LIN {X 0,Y 490.317,Z 298.891,A -85,B 0,C 180,E1 -6360.634,E2 -6360.634} C_VEL
LIN {X 0,Y 489.99,Z 352.828,A -85,B 0,C 180,E1 -6361.447,E2 -6361.447} C_VEL
LIN {X 0,Y 489.88,Z 362.097,A -85,B 0,C 180,E1 -6361.688,E2 -6361.688} C_VEL
LIN {X 0,Y 489.724,Z 372.302,A -85,B 0,C 180,E1 -6362.083,E2 -6362.083} C_VEL
LIN {X 0,Y 489.479,Z 384.149,A -85,B 0,C 180,E1 -6362.737,E2 -6362.737} C_VEL
LIN {X 0,Y 489.252,Z 392.699,A -85,B 0,C 180,E1 -6363.367,E2 -6363.367} C_VEL
LIN {X 0,Y 488.984,Z 399.772,A -85,B 0,C 180,E1 -6364,E2 -6364} C_VEL
LIN {X 0,Y 488.756,Z 406.629,A -85,B 0,C 180,E1 -6364.743,E2 -6364.743} C_VEL
LIN {X 0,Y 488.57,Z 412.949,A -85,B 0,C 180,E1 -6365.571,E2 -6365.571} C_VEL
LIN {X 0,Y 488.385,Z 418.571,A -85,B 0,C 180,E1 -6366.464,E2 -6366.464} C_VEL
LIN {X 0,Y 488.232,Z 423.172,A -85,B 0,C 180,E1 -6367.353,E2 -6367.353} C_VEL
LIN {X 0,Y 488.108,Z 427.721,A -85,B 0,C 180,E1 -6368.46,E2 -6368.46} C_VEL
LIN {X 0,Y 488.055,Z 430.624,A -85,B 0,C 180,E1 -6369.377,E2 -6369.377} C_VEL
LIN {X 0,Y 487.919,Z 433.524,A -85,B 0,C 180,E1 -6370.653,E2 -6370.653} C_VEL
LIN {X 0,Y 487.896,Z 435.193,A -85,B 0,C 180,E1 -6371.921,E2 -6371.921} C_VEL
LIN {X 0,Y 487.875,Z 435.589,A -85,B 0,C 180,E1 -6373.256,E2 -6373.256} C_VEL
LIN {X 0,Y 487.923,Z 435.219,A -85,B 0,C 180,E1 -6374.117,E2 -6374.117} C_VEL
LIN {X 0,Y 487.927,Z 434.243,A -85,B 0,C 180,E1 -6374.973,E2 -6374.973} C_VEL
LIN {X 0,Y 487.992,Z 431.831,A -85,B 0,C 180,E1 -6376.253,E2 -6376.253} C_VEL
LIN {X 0,Y 488.088,Z 428.018,A -85,B 0,C 180,E1 -6377.527,E2 -6377.527} C_VEL
LIN {X 0,Y 488.18,Z 424.744,A -85,B 0,C 180,E1 -6378.373,E2 -6378.373} C_VEL
LIN {X 0,Y 488.358,Z 419.564,A -85,B 0,C 180,E1 -6379.427,E2 -6379.427} C_VEL
LIN {X 0,Y 488.473,Z 414.514,A -85,B 0,C 180,E1 -6380.267,E2 -6380.267} C_VEL
LIN {X 0,Y 488.635,Z 408.418,A -85,B 0,C 180,E1 -6381.106,E2 -6381.106} C_VEL
LIN {X 0,Y 488.95,Z 401.875,A -85,B 0,C 180,E1 -6381.85,E2 -6381.85} C_VEL
LIN {X 0,Y 489.127,Z 394.255,A -85,B 0,C 180,E1 -6382.57,E2 -6382.57} C_VEL
LIN {X 0,Y 489.382,Z 386.064,A -85,B 0,C 180,E1 -6383.198,E2 -6383.198} C_VEL
LIN {X 0,Y 489.583,Z 377.622,A -85,B 0,C 180,E1 -6383.716,E2 -6383.716} C_VEL
LIN {X 0,Y 489.769,Z 367.721,A -85,B 0,C 180,E1 -6384.184,E2 -6384.184} C_VEL
LIN {X 0,Y 489.927,Z 355.422,A -85,B 0,C 180,E1 -6384.573,E2 -6384.573} C_VEL
LIN {X 0,Y 490.062,Z 334.881,A -85,B 0,C 180,E1 -6384.909,E2 -6384.909} C_VEL
LIN {X 0,Y 490.212,Z 286.553,A -85,B 0,C 180,E1 -6385.619,E2 -6385.619} C_VEL
LIN {X 0,Y 488.623,Z 277.035,A -85,B 0,C 180,E1 -6385.824,E2 -6385.824} C_VEL
LIN {X 0,Y 488.729,Z 264.417,A -85,B 0,C 180,E1 -6388.764,E2 -6388.764} C_VEL
LIN {X 0,Y 488.756,Z 259.415,A -85,B 0,C 180,E1 -6389.949,E2 -6389.949} C_VEL
LIN {X 0,Y 488.939,Z 259.395,A -85,B 0,C 180,E1 -6390.824,E2 -6390.824} C_VEL
LIN {X 0,Y 488.921,Z 259.391,A -85,B 0,C 180,E1 -6392.472,E2 -6392.472} C_VEL
LIN {X 0,Y 488.816,Z 259.406,A -85,B 0,C 180,E1 -6395.776,E2 -6395.776} C_VEL
LIN {X 0,Y 488.778,Z 259.408,A -85,B 0,C 180,E1 -6398.267,E2 -6398.267} C_VEL
LIN {X 0,Y 488.771,Z 259.414,A -85,B 0,C 180,E1 -6401.613,E2 -6401.613} C_VEL
LIN {X 0,Y 488.723,Z 259.419,A -85,B 0,C 180,E1 -6405.002,E2 -6405.002} C_VEL
LIN {X 0,Y 488.719,Z 259.415,A -85,B 0,C 180,E1 -6408.444,E2 -6408.444} C_VEL
LIN {X 0,Y 488.671,Z 259.425,A -85,B 0,C 180,E1 -6411.073,E2 -6411.073} C_VEL
LIN {X 0,Y 488.635,Z 259.43,A -85,B 0,C 180,E1 -6413.749,E2 -6413.749} C_VEL
LIN {X 0,Y 488.691,Z 259.421,A -85,B 0,C 180,E1 -6416.93,E2 -6416.93} C_VEL
LIN {X 0,Y 488.69,Z 259.419,A -85,B 0,C 180,E1 -6420.222,E2 -6420.222} C_VEL
LIN {X 0,Y 488.704,Z 259.426,A -85,B 0,C 180,E1 -6423.487,E2 -6423.487} C_VEL
LIN {X 0,Y 488.644,Z 259.425,A -85,B 0,C 180,E1 -6426.356,E2 -6426.356} C_VEL
LIN {X 0,Y 488.666,Z 259.426,A -85,B 0,C 180,E1 -6429.258,E2 -6429.258} C_VEL
LIN {X 0,Y 488.663,Z 259.423,A -85,B 0,C 180,E1 -6432.529,E2 -6432.529} C_VEL
LIN {X 0,Y 488.678,Z 259.424,A -85,B 0,C 180,E1 -6435.2,E2 -6435.2} C_VEL
LIN {X 0,Y 488.686,Z 259.42,A -85,B 0,C 180,E1 -6438.588,E2 -6438.588} C_VEL
LIN {X 0,Y 488.683,Z 259.421,A -85,B 0,C 180,E1 -6440.951,E2 -6440.951} C_VEL
LIN {X 0,Y 488.659,Z 259.43,A -85,B 0,C 180,E1 -6443.871,E2 -6443.871} C_VEL
LIN {X 0,Y 488.719,Z 259.416,A -85,B 0,C 180,E1 -6446.88,E2 -6446.88} C_VEL
LIN {X 0,Y 488.71,Z 259.426,A -85,B 0,C 180,E1 -6449.784,E2 -6449.784} C_VEL
LIN {X 0,Y 488.702,Z 259.419,A -85,B 0,C 180,E1 -6453.078,E2 -6453.078} C_VEL
LIN {X 0,Y 488.664,Z 259.426,A -85,B 0,C 180,E1 -6456.257,E2 -6456.257} C_VEL
LIN {X 0,Y 488.739,Z 259.415,A -85,B 0,C 180,E1 -6459.179,E2 -6459.179} C_VEL
LIN {X 0,Y 488.74,Z 259.418,A -85,B 0,C 180,E1 -6461.636,E2 -6461.636} C_VEL
LIN {X 0,Y 488.742,Z 259.419,A -85,B 0,C 180,E1 -6463.128,E2 -6463.128} C_VEL
LIN {X 0,Y 488.681,Z 269.044,A -85,B 0,C 180,E1 -6465.426,E2 -6465.426} C_VEL
LIN {X 0,Y 488.581,Z 277.029,A -85,B 0,C 180,E1 -6467.336,E2 -6467.336} C_VEL
LIN {X 0,Y 490.238,Z 287.915,A -85,B 0,C 180,E1 -6467.556,E2 -6467.556} C_VEL
LIN {X 0,Y 489.779,Z 353.824,A -85,B 0,C 180,E1 -6468.624,E2 -6468.624} C_VEL
LIN {X 0,Y 489.623,Z 363.696,A -85,B 0,C 180,E1 -6468.908,E2 -6468.908} C_VEL
LIN {X 0,Y 489.446,Z 373.101,A -85,B 0,C 180,E1 -6469.297,E2 -6469.297} C_VEL
LIN {X 0,Y 489.295,Z 383.431,A -85,B 0,C 180,E1 -6469.869,E2 -6469.869} C_VEL
LIN {X 0,Y 489.06,Z 393.321,A -85,B 0,C 180,E1 -6470.595,E2 -6470.595} C_VEL
LIN {X 0,Y 488.821,Z 401.151,A -85,B 0,C 180,E1 -6471.32,E2 -6471.32} C_VEL
LIN {X 0,Y 488.585,Z 408.483,A -85,B 0,C 180,E1 -6472.149,E2 -6472.149} C_VEL
LIN {X 0,Y 488.441,Z 413.629,A -85,B 0,C 180,E1 -6472.842,E2 -6472.842} C_VEL
LIN {X 0,Y 488.448,Z 418.403,A -85,B 0,C 180,E1 -6473.601,E2 -6473.601} C_VEL
LIN {X 0,Y 488.143,Z 423.728,A -85,B 0,C 180,E1 -6474.633,E2 -6474.633} C_VEL
LIN {X 0,Y 488.187,Z 427.167,A -85,B 0,C 180,E1 -6475.461,E2 -6475.461} C_VEL
LIN {X 0,Y 488.072,Z 431.112,A -85,B 0,C 180,E1 -6476.701,E2 -6476.701} C_VEL
LIN {X 0,Y 488.008,Z 432.994,A -85,B 0,C 180,E1 -6477.527,E2 -6477.527} C_VEL
LIN {X 0,Y 487.895,Z 434.357,A -85,B 0,C 180,E1 -6478.352,E2 -6478.352} C_VEL
LIN {X 0,Y 487.843,Z 435.219,A -85,B 0,C 180,E1 -6479.177,E2 -6479.177} C_VEL
LIN {X 0,Y 487.834,Z 435.549,A -85,B 0,C 180,E1 -6480.003,E2 -6480.003} C_VEL
LIN {X 0,Y 487.844,Z 435.297,A -85,B 0,C 180,E1 -6480.828,E2 -6480.828} C_VEL
LIN {X 0,Y 487.896,Z 434.545,A -85,B 0,C 180,E1 -6481.653,E2 -6481.653} C_VEL
LIN {X 0,Y 488.011,Z 433.293,A -85,B 0,C 180,E1 -6482.479,E2 -6482.479} C_VEL
LIN {X 0,Y 488.098,Z 430.396,A -85,B 0,C 180,E1 -6483.718,E2 -6483.718} C_VEL
LIN {X 0,Y 488.152,Z 426.21,A -85,B 0,C 180,E1 -6484.958,E2 -6484.958} C_VEL
LIN {X 0,Y 488.403,Z 420.333,A -85,B 0,C 180,E1 -6486.198,E2 -6486.198} C_VEL
LIN {X 0,Y 488.442,Z 414.686,A -85,B 0,C 180,E1 -6487.142,E2 -6487.142} C_VEL
LIN {X 0,Y 488.645,Z 407.893,A -85,B 0,C 180,E1 -6488.064,E2 -6488.064} C_VEL
LIN {X 0,Y 488.91,Z 399.373,A -85,B 0,C 180,E1 -6488.996,E2 -6488.996} C_VEL
LIN {X 0,Y 489.197,Z 389.497,A -85,B 0,C 180,E1 -6489.825,E2 -6489.825} C_VEL
LIN {X 0,Y 489.365,Z 381.81,A -85,B 0,C 180,E1 -6490.344,E2 -6490.344} C_VEL
LIN {X 0,Y 489.54,Z 372.044,A -85,B 0,C 180,E1 -6490.863,E2 -6490.863} C_VEL
LIN {X 0,Y 489.673,Z 360.611,A -85,B 0,C 180,E1 -6491.305,E2 -6491.305} C_VEL
LIN {X 0,Y 489.884,Z 348.005,A -85,B 0,C 180,E1 -6491.589,E2 -6491.589} C_VEL
LIN {X 0,Y 490.167,Z 286.104,A -85,B 0,C 180,E1 -6492.609,E2 -6492.609} C_VEL
LIN {X 0,Y 488.657,Z 277.687,A -85,B 0,C 180,E1 -6492.812,E2 -6492.812} C_VEL
LIN {X 0,Y 488.764,Z 264.596,A -85,B 0,C 180,E1 -6495.857,E2 -6495.857} C_VEL
LIN {X 0,Y 488.804,Z 259.414,A -85,B 0,C 180,E1 -6497.091,E2 -6497.091} C_VEL
LIN {X 0,Y 488.732,Z 259.423,A -85,B 0,C 180,E1 -6500.191,E2 -6500.191} C_VEL
LIN {X 0,Y 488.716,Z 259.419,A -85,B 0,C 180,E1 -6503.021,E2 -6503.021} C_VEL
LIN {X 0,Y 488.701,Z 259.421,A -85,B 0,C 180,E1 -6505.56,E2 -6505.56} C_VEL
LIN {X 0,Y 488.709,Z 259.423,A -85,B 0,C 180,E1 -6508.69,E2 -6508.69} C_VEL
LIN {X 0,Y 488.699,Z 259.42,A -85,B 0,C 180,E1 -6511.181,E2 -6511.181} C_VEL
LIN {X 0,Y 488.731,Z 259.42,A -85,B 0,C 180,E1 -6514.115,E2 -6514.115} C_VEL
LIN {X 0,Y 488.678,Z 259.423,A -85,B 0,C 180,E1 -6517.161,E2 -6517.161} C_VEL
LIN {X 0,Y 488.701,Z 259.426,A -85,B 0,C 180,E1 -6520.342,E2 -6520.342} C_VEL
LIN {X 0,Y 488.686,Z 259.42,A -85,B 0,C 180,E1 -6523.656,E2 -6523.656} C_VEL
LIN {X 0,Y 488.686,Z 259.425,A -85,B 0,C 180,E1 -6526.345,E2 -6526.345} C_VEL
LIN {X 0,Y 488.711,Z 259.417,A -85,B 0,C 180,E1 -6529.674,E2 -6529.674} C_VEL
LIN {X 0,Y 488.677,Z 259.425,A -85,B 0,C 180,E1 -6532.841,E2 -6532.841} C_VEL
LIN {X 0,Y 488.727,Z 259.415,A -85,B 0,C 180,E1 -6535.887,E2 -6535.887} C_VEL
LIN {X 0,Y 488.698,Z 259.425,A -85,B 0,C 180,E1 -6538.82,E2 -6538.82} C_VEL
LIN {X 0,Y 488.748,Z 259.414,A -85,B 0,C 180,E1 -6541.671,E2 -6541.671} C_VEL
LIN {X 0,Y 488.759,Z 259.413,A -85,B 0,C 180,E1 -6543.528,E2 -6543.528} C_VEL
LIN {X 0,Y 488.777,Z 259.557,A -85,B 0,C 180,E1 -6546.09,E2 -6546.09} C_VEL
LIN {X 0,Y 489.904,Z 266.437,A -85,B 0,C 180,E1 -6547.434,E2 -6547.434} C_VEL
LIN {X 0,Y 489.528,Z 279.387,A -85,B 0,C 180,E1 -6549.845,E2 -6549.845} C_VEL
LIN {X 0,Y 489.111,Z 294.638,A -85,B 0,C 180,E1 -6552.653,E2 -6552.653} C_VEL
LIN {X 0,Y 488.736,Z 310.996,A -85,B 0,C 180,E1 -6555.637,E2 -6555.637} C_VEL
LIN {X 0,Y 488.559,Z 319.87,A -85,B 0,C 180,E1 -6557.219,E2 -6557.219} C_VEL
LIN {X 0,Y 490.207,Z 335.706,A -85,B 0,C 180,E1 -6557.494,E2 -6557.494} C_VEL
LIN {X 0,Y 489.919,Z 397.001,A -85,B 0,C 180,E1 -6558.414,E2 -6558.414} C_VEL
LIN {X 0,Y 489.685,Z 406.883,A -85,B 0,C 180,E1 -6558.671,E2 -6558.671} C_VEL
LIN {X 0,Y 489.424,Z 417.462,A -85,B 0,C 180,E1 -6559.084,E2 -6559.084} C_VEL
LIN {X 0,Y 489.203,Z 427.831,A -85,B 0,C 180,E1 -6559.655,E2 -6559.655} C_VEL
LIN {X 0,Y 488.94,Z 436.482,A -85,B 0,C 180,E1 -6560.276,E2 -6560.276} C_VEL
LIN {X 0,Y 488.705,Z 444.617,A -85,B 0,C 180,E1 -6561.002,E2 -6561.002} C_VEL
LIN {X 0,Y 488.479,Z 451.337,A -85,B 0,C 180,E1 -6561.728,E2 -6561.728} C_VEL
LIN {X 0,Y 488.304,Z 457.716,A -85,B 0,C 180,E1 -6562.557,E2 -6562.557} C_VEL
LIN {X 0,Y 488.185,Z 463.018,A -85,B 0,C 180,E1 -6563.386,E2 -6563.386} C_VEL
LIN {X 0,Y 488.095,Z 467.44,A -85,B 0,C 180,E1 -6564.215,E2 -6564.215} C_VEL
LIN {X 0,Y 487.95,Z 472.646,A -85,B 0,C 180,E1 -6565.456,E2 -6565.456} C_VEL
LIN {X 0,Y 487.986,Z 476.475,A -85,B 0,C 180,E1 -6566.697,E2 -6566.697} C_VEL
LIN {X 0,Y 487.937,Z 478.234,A -85,B 0,C 180,E1 -6567.523,E2 -6567.523} C_VEL
LIN {X 0,Y 487.892,Z 479.493,A -85,B 0,C 180,E1 -6568.349,E2 -6568.349} C_VEL
LIN {X 0,Y 487.837,Z 480.275,A -85,B 0,C 180,E1 -6569.174,E2 -6569.174} C_VEL
LIN {X 0,Y 487.828,Z 480.568,A -85,B 0,C 180,E1 -6570,E2 -6570} C_VEL
LIN {X 0,Y 487.837,Z 480.267,A -85,B 0,C 180,E1 -6570.825,E2 -6570.825} C_VEL
LIN {X 0,Y 487.892,Z 479.481,A -85,B 0,C 180,E1 -6571.651,E2 -6571.651} C_VEL
LIN {X 0,Y 487.937,Z 478.218,A -85,B 0,C 180,E1 -6572.476,E2 -6572.476} C_VEL
LIN {X 0,Y 488.006,Z 475.293,A -85,B 0,C 180,E1 -6573.716,E2 -6573.716} C_VEL
LIN {X 0,Y 487.95,Z 472.624,A -85,B 0,C 180,E1 -6574.543,E2 -6574.543} C_VEL
LIN {X 0,Y 488.095,Z 467.413,A -85,B 0,C 180,E1 -6575.785,E2 -6575.785} C_VEL
LIN {X 0,Y 488.278,Z 460.55,A -85,B 0,C 180,E1 -6577.027,E2 -6577.027} C_VEL
LIN {X 0,Y 488.408,Z 453.049,A -85,B 0,C 180,E1 -6578.065,E2 -6578.065} C_VEL
LIN {X 0,Y 488.685,Z 445.662,A -85,B 0,C 180,E1 -6578.893,E2 -6578.893} C_VEL
LIN {X 0,Y 488.934,Z 437.755,A -85,B 0,C 180,E1 -6579.619,E2 -6579.619} C_VEL
LIN {X 0,Y 489.148,Z 429.404,A -85,B 0,C 180,E1 -6580.242,E2 -6580.242} C_VEL
LIN {X 0,Y 489.419,Z 418.752,A -85,B 0,C 180,E1 -6580.864,E2 -6580.864} C_VEL
LIN {X 0,Y 489.675,Z 407.189,A -85,B 0,C 180,E1 -6581.329,E2 -6581.329} C_VEL
LIN {X 0,Y 489.897,Z 397.546,A -85,B 0,C 180,E1 -6581.586,E2 -6581.586} C_VEL
LIN {X 0,Y 490.181,Z 349.611,A -85,B 0,C 180,E1 -6582.312,E2 -6582.312} C_VEL
LIN {X 0,Y 490.091,Z 332.403,A -85,B 0,C 180,E1 -6582.569,E2 -6582.569} C_VEL
LIN {X 0,Y 488.567,Z 319.475,A -85,B 0,C 180,E1 -6582.807,E2 -6582.807} C_VEL
LIN {X 0,Y 488.922,Z 302.661,A -85,B 0,C 180,E1 -6585.85,E2 -6585.85} C_VEL
LIN {X 0,Y 489.44,Z 283.877,A -85,B 0,C 180,E1 -6589.285,E2 -6589.285} C_VEL
LIN {X 0,Y 489.897,Z 267.404,A -85,B 0,C 180,E1 -6592.344,E2 -6592.344} C_VEL
LIN {X 0,Y 488.77,Z 259.552,A -85,B 0,C 180,E1 -6593.882,E2 -6593.882} C_VEL
LIN {X 0,Y 488.797,Z 259.413,A -85,B 0,C 180,E1 -6596.943,E2 -6596.943} C_VEL
LIN {X 0,Y 488.713,Z 259.417,A -85,B 0,C 180,E1 -6600.362,E2 -6600.362} C_VEL
LIN {X 0,Y 488.716,Z 259.425,A -85,B 0,C 180,E1 -6603.479,E2 -6603.479} C_VEL
LIN {X 0,Y 488.687,Z 259.418,A -85,B 0,C 180,E1 -6606.354,E2 -6606.354} C_VEL
LIN {X 0,Y 488.706,Z 259.424,A -85,B 0,C 180,E1 -6609.254,E2 -6609.254} C_VEL
LIN {X 0,Y 488.695,Z 259.419,A -85,B 0,C 180,E1 -6612.525,E2 -6612.525} C_VEL
LIN {X 0,Y 488.708,Z 259.42,A -85,B 0,C 180,E1 -6615.196,E2 -6615.196} C_VEL
LIN {X 0,Y 488.701,Z 259.418,A -85,B 0,C 180,E1 -6618.582,E2 -6618.582} C_VEL
LIN {X 0,Y 488.706,Z 259.417,A -85,B 0,C 180,E1 -6620.947,E2 -6620.947} C_VEL
LIN {X 0,Y 488.683,Z 259.423,A -85,B 0,C 180,E1 -6623.867,E2 -6623.867} C_VEL
LIN {X 0,Y 488.741,Z 259.413,A -85,B 0,C 180,E1 -6626.876,E2 -6626.876} C_VEL
LIN {X 0,Y 488.728,Z 259.421,A -85,B 0,C 180,E1 -6629.779,E2 -6629.779} C_VEL
LIN {X 0,Y 488.731,Z 259.414,A -85,B 0,C 180,E1 -6633.07,E2 -6633.07} C_VEL
LIN {X 0,Y 488.717,Z 259.418,A -85,B 0,C 180,E1 -6635.351,E2 -6635.351} C_VEL
LIN {X 0,Y 488.703,Z 259.419,A -85,B 0,C 180,E1 -6638.041,E2 -6638.041} C_VEL
LIN {X 0,Y 488.745,Z 259.412,A -85,B 0,C 180,E1 -6640.685,E2 -6640.685} C_VEL
LIN {X 0,Y 488.765,Z 259.412,A -85,B 0,C 180,E1 -6644.143,E2 -6644.143} C_VEL
LIN {X 0,Y 488.732,Z 259.413,A -85,B 0,C 180,E1 -6646.696,E2 -6646.696} C_VEL
LIN {X 0,Y 488.738,Z 259.408,A -85,B 0,C 180,E1 -6649.224,E2 -6649.224} C_VEL
LIN {X 0,Y 488.866,Z 259.396,A -85,B 0,C 180,E1 -6652.564,E2 -6652.564} C_VEL
LIN {X 0,Y 488.81,Z 259.399,A -85,B 0,C 180,E1 -6655.049,E2 -6655.049} C_VEL
LIN {X 0,Y 488.954,Z 259.387,A -85,B 0,C 180,E1 -6657.526,E2 -6657.526} C_VEL
LIN {X 0,Y 488.97,Z 259.386,A -85,B 0,C 180,E1 -6659.997,E2 -6659.997} C_VEL
LIN {X 0,Y 488.953,Z 259.389,A -85,B 0,C 180,E1 -6662.469,E2 -6662.469} C_VEL
LIN {X 0,Y 488.833,Z 259.4,A -85,B 0,C 180,E1 -6665.773,E2 -6665.773} C_VEL
LIN {X 0,Y 488.783,Z 259.415,A -85,B 0,C 180,E1 -6668.264,E2 -6668.264} C_VEL
LIN {X 0,Y 488.801,Z 259.404,A -85,B 0,C 180,E1 -6671.609,E2 -6671.609} C_VEL
LIN {X 0,Y 488.755,Z 259.409,A -85,B 0,C 180,E1 -6674.997,E2 -6674.997} C_VEL
LIN {X 0,Y 488.738,Z 259.42,A -85,B 0,C 180,E1 -6678.439,E2 -6678.439} C_VEL
LIN {X 0,Y 488.697,Z 259.418,A -85,B 0,C 180,E1 -6681.068,E2 -6681.068} C_VEL
LIN {X 0,Y 488.677,Z 259.422,A -85,B 0,C 180,E1 -6683.742,E2 -6683.742} C_VEL
LIN {X 0,Y 488.779,Z 259.41,A -85,B 0,C 180,E1 -6686.94,E2 -6686.94} C_VEL
LIN {X 0,Y 488.694,Z 259.426,A -85,B 0,C 180,E1 -6690.36,E2 -6690.36} C_VEL
LIN {X 0,Y 488.718,Z 259.416,A -85,B 0,C 180,E1 -6693.481,E2 -6693.481} C_VEL
LIN {X 0,Y 488.668,Z 259.422,A -85,B 0,C 180,E1 -6696.352,E2 -6696.352} C_VEL
LIN {X 0,Y 488.68,Z 259.421,A -85,B 0,C 180,E1 -6699.251,E2 -6699.251} C_VEL
LIN {X 0,Y 488.712,Z 259.424,A -85,B 0,C 180,E1 -6702.518,E2 -6702.518} C_VEL
LIN {X 0,Y 488.677,Z 259.423,A -85,B 0,C 180,E1 -6705.973,E2 -6705.973} C_VEL
LIN {X 0,Y 488.701,Z 259.426,A -85,B 0,C 180,E1 -6708.584,E2 -6708.584} C_VEL
LIN {X 0,Y 488.72,Z 259.423,A -85,B 0,C 180,E1 -6710.938,E2 -6710.938} C_VEL
LIN {X 0,Y 488.658,Z 259.427,A -85,B 0,C 180,E1 -6713.866,E2 -6713.866} C_VEL
LIN {X 0,Y 488.653,Z 259.467,A -85,B 0,C 180,E1 -6716.329,E2 -6716.329} C_VEL
LIN {X 0,Y 488.62,Z 270.599,A -85,B 0,C 180,E1 -6718.815,E2 -6718.815} C_VEL
LIN {X 0,Y 488.642,Z 277.255,A -85,B 0,C 180,E1 -6720.264,E2 -6720.264} C_VEL
LIN {X 0,Y 490.394,Z 287.787,A -85,B 0,C 180,E1 -6720.471,E2 -6720.471} C_VEL
LIN {X 0,Y 490.317,Z 298.891,A -85,B 0,C 180,E1 -6720.634,E2 -6720.634} C_VEL
LIN {X 0,Y 489.629,Z 304.733,A -85,B 0,C 180,E1 -6720.701,E2 -6720.701} C_VEL
LIN {X 0,Y 483.957,Z 323.717,A -85,B 0,C 180,E1 -6720.826,E2 -6720.826} C_VEL
LIN {X 0,Y 483.262,Z 329.559,A -85,B 0,C 180,E1 -6720.894,E2 -6720.894} C_VEL
LIN {X 0,Y 483.068,Z 354.101,A -85,B 0,C 180,E1 -6721.287,E2 -6721.287} C_VEL
LIN {X 0,Y 482.918,Z 365.022,A -85,B 0,C 180,E1 -6721.595,E2 -6721.595} C_VEL
LIN {X 0,Y 482.718,Z 376.658,A -85,B 0,C 180,E1 -6722.114,E2 -6722.114} C_VEL
LIN {X 0,Y 482.488,Z 385.923,A -85,B 0,C 180,E1 -6722.68,E2 -6722.68} C_VEL
LIN {X 0,Y 482.268,Z 393.536,A -85,B 0,C 180,E1 -6723.261,E2 -6723.261} C_VEL
LIN {X 0,Y 481.956,Z 400.889,A -85,B 0,C 180,E1 -6723.942,E2 -6723.942} C_VEL
LIN {X 0,Y 481.709,Z 408.076,A -85,B 0,C 180,E1 -6724.754,E2 -6724.754} C_VEL
LIN {X 0,Y 481.507,Z 414.571,A -85,B 0,C 180,E1 -6725.649,E2 -6725.649} C_VEL
LIN {X 0,Y 481.267,Z 421.209,A -85,B 0,C 180,E1 -6726.779,E2 -6726.779} C_VEL
LIN {X 0,Y 481.065,Z 427.118,A -85,B 0,C 180,E1 -6728.128,E2 -6728.128} C_VEL
LIN {X 0,Y 480.991,Z 430.728,A -85,B 0,C 180,E1 -6729.237,E2 -6729.237} C_VEL
LIN {X 0,Y 480.85,Z 433.361,A -85,B 0,C 180,E1 -6730.357,E2 -6730.357} C_VEL
LIN {X 0,Y 480.815,Z 435.422,A -85,B 0,C 180,E1 -6731.807,E2 -6731.807} C_VEL
LIN {X 0,Y 480.775,Z 435.972,A -85,B 0,C 180,E1 -6733.001,E2 -6733.001} C_VEL
LIN {X 0,Y 480.831,Z 435.672,A -85,B 0,C 180,E1 -6733.877,E2 -6733.877} C_VEL
LIN {X 0,Y 480.836,Z 434.856,A -85,B 0,C 180,E1 -6734.747,E2 -6734.747} C_VEL
LIN {X 0,Y 480.866,Z 433.526,A -85,B 0,C 180,E1 -6735.614,E2 -6735.614} C_VEL
LIN {X 0,Y 480.959,Z 430.484,A -85,B 0,C 180,E1 -6736.909,E2 -6736.909} C_VEL
LIN {X 0,Y 481.093,Z 426.132,A -85,B 0,C 180,E1 -6738.199,E2 -6738.199} C_VEL
LIN {X 0,Y 481.303,Z 420.07,A -85,B 0,C 180,E1 -6739.483,E2 -6739.483} C_VEL
LIN {X 0,Y 481.428,Z 415.056,A -85,B 0,C 180,E1 -6740.336,E2 -6740.336} C_VEL
LIN {X 0,Y 481.607,Z 408.995,A -85,B 0,C 180,E1 -6741.186,E2 -6741.186} C_VEL
LIN {X 0,Y 481.968,Z 401.571,A -85,B 0,C 180,E1 -6742.037,E2 -6742.037} C_VEL
LIN {X 0,Y 482.111,Z 395.2,A -85,B 0,C 180,E1 -6742.649,E2 -6742.649} C_VEL
LIN {X 0,Y 482.353,Z 388.181,A -85,B 0,C 180,E1 -6743.213,E2 -6743.213} C_VEL
LIN {X 0,Y 482.554,Z 380.339,A -85,B 0,C 180,E1 -6743.729,E2 -6743.729} C_VEL
LIN {X 0,Y 482.718,Z 371.145,A -85,B 0,C 180,E1 -6744.203,E2 -6744.203} C_VEL
LIN {X 0,Y 482.934,Z 362.156,A -85,B 0,C 180,E1 -6744.546,E2 -6744.546} C_VEL
LIN {X 0,Y 483.02,Z 353.222,A -85,B 0,C 180,E1 -6744.783,E2 -6744.783} C_VEL
LIN {X 0,Y 483.265,Z 287.076,A -85,B 0,C 180,E1 -6745.791,E2 -6745.791} C_VEL
LIN {X 0,Y 481.559,Z 277.317,A -85,B 0,C 180,E1 -6745.999,E2 -6745.999} C_VEL
LIN {X 0,Y 481.702,Z 265.598,A -85,B 0,C 180,E1 -6748.746,E2 -6748.746} C_VEL
LIN {X 0,Y 481.724,Z 260.291,A -85,B 0,C 180,E1 -6750,E2 -6750} C_VEL
LIN {X 0,Y 481.776,Z 260.284,A -85,B 0,C 180,E1 -6751.672,E2 -6751.672} C_VEL
LIN {X 0,Y 481.889,Z 260.267,A -85,B 0,C 180,E1 -6752.508,E2 -6752.508} C_VEL
LIN {X 0,Y 481.776,Z 260.282,A -85,B 0,C 180,E1 -6755.861,E2 -6755.861} C_VEL
LIN {X 0,Y 481.724,Z 260.287,A -85,B 0,C 180,E1 -6758.389,E2 -6758.389} C_VEL
LIN {X 0,Y 481.715,Z 260.291,A -85,B 0,C 180,E1 -6761.786,E2 -6761.786} C_VEL
LIN {X 0,Y 481.705,Z 260.296,A -85,B 0,C 180,E1 -6765.226,E2 -6765.226} C_VEL
LIN {X 0,Y 481.676,Z 260.294,A -85,B 0,C 180,E1 -6768.723,E2 -6768.723} C_VEL
LIN {X 0,Y 481.61,Z 260.31,A -85,B 0,C 180,E1 -6771.397,E2 -6771.397} C_VEL
LIN {X 0,Y 481.614,Z 260.301,A -85,B 0,C 180,E1 -6774.117,E2 -6774.117} C_VEL
LIN {X 0,Y 481.661,Z 260.299,A -85,B 0,C 180,E1 -6777.129,E2 -6777.129} C_VEL
LIN {X 0,Y 481.64,Z 260.302,A -85,B 0,C 180,E1 -6779.744,E2 -6779.744} C_VEL
LIN {X 0,Y 481.641,Z 260.297,A -85,B 0,C 180,E1 -6782.677,E2 -6782.677} C_VEL
LIN {X 0,Y 481.602,Z 260.308,A -85,B 0,C 180,E1 -6785.713,E2 -6785.713} C_VEL
LIN {X 0,Y 481.638,Z 260.299,A -85,B 0,C 180,E1 -6788.863,E2 -6788.863} C_VEL
LIN {X 0,Y 481.615,Z 260.302,A -85,B 0,C 180,E1 -6792.165,E2 -6792.165} C_VEL
LIN {X 0,Y 481.632,Z 260.306,A -85,B 0,C 180,E1 -6795.545,E2 -6795.545} C_VEL
LIN {X 0,Y 481.635,Z 260.299,A -85,B 0,C 180,E1 -6798.961,E2 -6798.961} C_VEL
LIN {X 0,Y 481.634,Z 260.303,A -85,B 0,C 180,E1 -6801.996,E2 -6801.996} C_VEL
LIN {X 0,Y 481.668,Z 260.297,A -85,B 0,C 180,E1 -6805.321,E2 -6805.321} C_VEL
LIN {X 0,Y 481.629,Z 260.301,A -85,B 0,C 180,E1 -6808.315,E2 -6808.315} C_VEL
LIN {X 0,Y 481.661,Z 260.297,A -85,B 0,C 180,E1 -6811.22,E2 -6811.22} C_VEL
LIN {X 0,Y 481.644,Z 260.303,A -85,B 0,C 180,E1 -6814.044,E2 -6814.044} C_VEL
LIN {X 0,Y 481.665,Z 260.295,A -85,B 0,C 180,E1 -6816.815,E2 -6816.815} C_VEL
LIN {X 0,Y 481.687,Z 260.296,A -85,B 0,C 180,E1 -6819.506,E2 -6819.506} C_VEL
LIN {X 0,Y 481.674,Z 260.299,A -85,B 0,C 180,E1 -6822.161,E2 -6822.161} C_VEL
LIN {X 0,Y 481.691,Z 260.407,A -85,B 0,C 180,E1 -6823.119,E2 -6823.119} C_VEL
LIN {X 0,Y 481.603,Z 270.901,A -85,B 0,C 180,E1 -6825.639,E2 -6825.639} C_VEL
LIN {X 0,Y 481.576,Z 277.482,A -85,B 0,C 180,E1 -6827.165,E2 -6827.165} C_VEL
LIN {X 0,Y 483.254,Z 287.503,A -85,B 0,C 180,E1 -6827.376,E2 -6827.376} C_VEL
LIN {X 0,Y 482.803,Z 354.23,A -85,B 0,C 180,E1 -6828.484,E2 -6828.484} C_VEL
LIN {X 0,Y 482.621,Z 364.045,A -85,B 0,C 180,E1 -6828.772,E2 -6828.772} C_VEL
LIN {X 0,Y 482.428,Z 373.972,A -85,B 0,C 180,E1 -6829.193,E2 -6829.193} C_VEL
LIN {X 0,Y 482.253,Z 384.99,A -85,B 0,C 180,E1 -6829.825,E2 -6829.825} C_VEL
LIN {X 0,Y 482.036,Z 394.515,A -85,B 0,C 180,E1 -6830.563,E2 -6830.563} C_VEL
LIN {X 0,Y 481.813,Z 401.22,A -85,B 0,C 180,E1 -6831.193,E2 -6831.193} C_VEL
LIN {X 0,Y 481.558,Z 408.597,A -85,B 0,C 180,E1 -6832.034,E2 -6832.034} C_VEL
LIN {X 0,Y 481.377,Z 414.967,A -85,B 0,C 180,E1 -6832.916,E2 -6832.916} C_VEL
LIN {X 0,Y 481.3,Z 420.899,A -85,B 0,C 180,E1 -6833.926,E2 -6833.926} C_VEL
LIN {X 0,Y 481.055,Z 425.836,A -85,B 0,C 180,E1 -6834.974,E2 -6834.974} C_VEL
LIN {X 0,Y 481.029,Z 430.23,A -85,B 0,C 180,E1 -6836.233,E2 -6836.233} C_VEL
LIN {X 0,Y 480.918,Z 433.279,A -85,B 0,C 180,E1 -6837.49,E2 -6837.49} C_VEL
LIN {X 0,Y 480.828,Z 434.654,A -85,B 0,C 180,E1 -6838.328,E2 -6838.328} C_VEL
LIN {X 0,Y 480.768,Z 435.529,A -85,B 0,C 180,E1 -6839.165,E2 -6839.165} C_VEL
LIN {X 0,Y 480.757,Z 435.865,A -85,B 0,C 180,E1 -6840.003,E2 -6840.003} C_VEL
LIN {X 0,Y 480.769,Z 435.617,A -85,B 0,C 180,E1 -6840.84,E2 -6840.84} C_VEL
LIN {X 0,Y 480.828,Z 434.868,A -85,B 0,C 180,E1 -6841.678,E2 -6841.678} C_VEL
LIN {X 0,Y 480.951,Z 433.615,A -85,B 0,C 180,E1 -6842.515,E2 -6842.515} C_VEL
LIN {X 0,Y 481.028,Z 430.713,A -85,B 0,C 180,E1 -6843.772,E2 -6843.772} C_VEL
LIN {X 0,Y 481.072,Z 426.517,A -85,B 0,C 180,E1 -6845.031,E2 -6845.031} C_VEL
LIN {X 0,Y 481.368,Z 420.644,A -85,B 0,C 180,E1 -6846.284,E2 -6846.284} C_VEL
LIN {X 0,Y 481.377,Z 415.994,A -85,B 0,C 180,E1 -6847.089,E2 -6847.089} C_VEL
LIN {X 0,Y 481.571,Z 409.815,A -85,B 0,C 180,E1 -6847.972,E2 -6847.972} C_VEL
LIN {X 0,Y 481.805,Z 402.643,A -85,B 0,C 180,E1 -6848.813,E2 -6848.813} C_VEL
LIN {X 0,Y 482.065,Z 393.822,A -85,B 0,C 180,E1 -6849.654,E2 -6849.654} C_VEL
LIN {X 0,Y 482.385,Z 383.838,A -85,B 0,C 180,E1 -6850.389,E2 -6850.389} C_VEL
LIN {X 0,Y 482.549,Z 374.554,A -85,B 0,C 180,E1 -6850.916,E2 -6850.916} C_VEL
LIN {X 0,Y 482.687,Z 365.401,A -85,B 0,C 180,E1 -6851.312,E2 -6851.312} C_VEL
LIN {X 0,Y 482.8,Z 355.976,A -85,B 0,C 180,E1 -6851.602,E2 -6851.602} C_VEL
LIN {X 0,Y 483.059,Z 333.092,A -85,B 0,C 180,E1 -6852.013,E2 -6852.013} C_VEL
LIN {X 0,Y 483.316,Z 287.11,A -85,B 0,C 180,E1 -6852.794,E2 -6852.794} C_VEL
LIN {X 0,Y 481.668,Z 278.03,A -85,B 0,C 180,E1 -6853.026,E2 -6853.026} C_VEL
LIN {X 0,Y 481.766,Z 264.867,A -85,B 0,C 180,E1 -6856.094,E2 -6856.094} C_VEL
LIN {X 0,Y 481.782,Z 260.289,A -85,B 0,C 180,E1 -6857.183,E2 -6857.183} C_VEL
LIN {X 0,Y 481.703,Z 260.298,A -85,B 0,C 180,E1 -6860.499,E2 -6860.499} C_VEL
LIN {X 0,Y 481.673,Z 260.296,A -85,B 0,C 180,E1 -6863.203,E2 -6863.203} C_VEL
LIN {X 0,Y 481.654,Z 260.302,A -85,B 0,C 180,E1 -6865.962,E2 -6865.962} C_VEL
LIN {X 0,Y 481.662,Z 260.299,A -85,B 0,C 180,E1 -6868.899,E2 -6868.899} C_VEL
LIN {X 0,Y 481.664,Z 260.301,A -85,B 0,C 180,E1 -6872.19,E2 -6872.19} C_VEL
LIN {X 0,Y 481.666,Z 260.296,A -85,B 0,C 180,E1 -6875.204,E2 -6875.204} C_VEL
LIN {X 0,Y 481.674,Z 260.298,A -85,B 0,C 180,E1 -6878.861,E2 -6878.861} C_VEL
LIN {X 0,Y 481.648,Z 260.301,A -85,B 0,C 180,E1 -6882.162,E2 -6882.162} C_VEL
LIN {X 0,Y 481.662,Z 260.295,A -85,B 0,C 180,E1 -6885.543,E2 -6885.543} C_VEL
LIN {X 0,Y 481.655,Z 260.3,A -85,B 0,C 180,E1 -6888.958,E2 -6888.958} C_VEL
LIN {X 0,Y 481.656,Z 260.298,A -85,B 0,C 180,E1 -6891.994,E2 -6891.994} C_VEL
LIN {X 0,Y 481.69,Z 260.293,A -85,B 0,C 180,E1 -6895.318,E2 -6895.318} C_VEL
LIN {X 0,Y 481.65,Z 260.301,A -85,B 0,C 180,E1 -6898.312,E2 -6898.312} C_VEL
LIN {X 0,Y 481.704,Z 260.294,A -85,B 0,C 180,E1 -6901.219,E2 -6901.219} C_VEL
LIN {X 0,Y 481.695,Z 260.293,A -85,B 0,C 180,E1 -6904.042,E2 -6904.042} C_VEL
LIN {X 0,Y 481.72,Z 260.326,A -85,B 0,C 180,E1 -6905.946,E2 -6905.946} C_VEL
LIN {X 0,Y 482.876,Z 267.205,A -85,B 0,C 180,E1 -6907.313,E2 -6907.313} C_VEL
LIN {X 0,Y 482.611,Z 277.835,A -85,B 0,C 180,E1 -6909.323,E2 -6909.323} C_VEL
LIN {X 0,Y 482.156,Z 293.087,A -85,B 0,C 180,E1 -6912.175,E2 -6912.175} C_VEL
LIN {X 0,Y 481.715,Z 310.63,A -85,B 0,C 180,E1 -6915.423,E2 -6915.423} C_VEL
LIN {X 0,Y 481.527,Z 319.299,A -85,B 0,C 180,E1 -6917.019,E2 -6917.019} C_VEL
LIN {X 0,Y 483.263,Z 336.852,A -85,B 0,C 180,E1 -6917.341,E2 -6917.341} C_VEL
LIN {X 0,Y 482.955,Z 396.427,A -85,B 0,C 180,E1 -6918.245,E2 -6918.245} C_VEL
LIN {X 0,Y 482.727,Z 405.566,A -85,B 0,C 180,E1 -6918.479,E2 -6918.479} C_VEL
LIN {X 0,Y 482.52,Z 414.598,A -85,B 0,C 180,E1 -6918.819,E2 -6918.819} C_VEL
LIN {X 0,Y 482.27,Z 423.891,A -85,B 0,C 180,E1 -6919.292,E2 -6919.292} C_VEL
LIN {X 0,Y 482.001,Z 433.457,A -85,B 0,C 180,E1 -6919.923,E2 -6919.923} C_VEL
LIN {X 0,Y 481.693,Z 443.216,A -85,B 0,C 180,E1 -6920.764,E2 -6920.764} C_VEL
LIN {X 0,Y 481.417,Z 450.971,A -85,B 0,C 180,E1 -6921.605,E2 -6921.605} C_VEL
LIN {X 0,Y 481.235,Z 457.357,A -85,B 0,C 180,E1 -6922.447,E2 -6922.447} C_VEL
LIN {X 0,Y 481.087,Z 463.352,A -85,B 0,C 180,E1 -6923.411,E2 -6923.411} C_VEL
LIN {X 0,Y 480.99,Z 469.019,A -85,B 0,C 180,E1 -6924.55,E2 -6924.55} C_VEL
LIN {X 0,Y 480.85,Z 473.794,A -85,B 0,C 180,E1 -6925.809,E2 -6925.809} C_VEL
LIN {X 0,Y 480.915,Z 476.138,A -85,B 0,C 180,E1 -6926.649,E2 -6926.649} C_VEL
LIN {X 0,Y 480.85,Z 477.9,A -85,B 0,C 180,E1 -6927.487,E2 -6927.487} C_VEL
LIN {X 0,Y 480.824,Z 479.163,A -85,B 0,C 180,E1 -6928.325,E2 -6928.325} C_VEL
LIN {X 0,Y 480.763,Z 479.948,A -85,B 0,C 180,E1 -6929.162,E2 -6929.162} C_VEL
LIN {X 0,Y 480.751,Z 480.242,A -85,B 0,C 180,E1 -6930,E2 -6930} C_VEL
LIN {X 0,Y 480.763,Z 479.942,A -85,B 0,C 180,E1 -6930.837,E2 -6930.837} C_VEL
LIN {X 0,Y 480.824,Z 479.159,A -85,B 0,C 180,E1 -6931.675,E2 -6931.675} C_VEL
LIN {X 0,Y 480.85,Z 477.898,A -85,B 0,C 180,E1 -6932.513,E2 -6932.513} C_VEL
LIN {X 0,Y 480.926,Z 474.974,A -85,B 0,C 180,E1 -6933.77,E2 -6933.77} C_VEL
LIN {X 0,Y 480.868,Z 472.307,A -85,B 0,C 180,E1 -6934.61,E2 -6934.61} C_VEL
LIN {X 0,Y 481,Z 467.097,A -85,B 0,C 180,E1 -6935.87,E2 -6935.87} C_VEL
LIN {X 0,Y 481.172,Z 461.497,A -85,B 0,C 180,E1 -6936.921,E2 -6936.921} C_VEL
LIN {X 0,Y 481.302,Z 454.449,A -85,B 0,C 180,E1 -6937.974,E2 -6937.974} C_VEL
LIN {X 0,Y 481.621,Z 446.387,A -85,B 0,C 180,E1 -6938.919,E2 -6938.919} C_VEL
LIN {X 0,Y 481.89,Z 438.696,A -85,B 0,C 180,E1 -6939.655,E2 -6939.655} C_VEL
LIN {X 0,Y 482.095,Z 430.632,A -85,B 0,C 180,E1 -6940.287,E2 -6940.287} C_VEL
LIN {X 0,Y 482.322,Z 422.296,A -85,B 0,C 180,E1 -6940.813,E2 -6940.813} C_VEL
LIN {X 0,Y 482.55,Z 413.809,A -85,B 0,C 180,E1 -6941.233,E2 -6941.233} C_VEL
LIN {X 0,Y 482.773,Z 404.555,A -85,B 0,C 180,E1 -6941.573,E2 -6941.573} C_VEL
LIN {X 0,Y 483.063,Z 394.641,A -85,B 0,C 180,E1 -6941.812,E2 -6941.812} C_VEL
LIN {X 0,Y 483.216,Z 333.364,A -85,B 0,C 180,E1 -6942.74,E2 -6942.74} C_VEL
LIN {X 0,Y 481.539,Z 319.049,A -85,B 0,C 180,E1 -6943.022,E2 -6943.022} C_VEL
LIN {X 0,Y 481.893,Z 302.38,A -85,B 0,C 180,E1 -6946.087,E2 -6946.087} C_VEL
LIN {X 0,Y 482.473,Z 283.615,A -85,B 0,C 180,E1 -6949.574,E2 -6949.574} C_VEL
LIN {X 0,Y 482.934,Z 268.333,A -85,B 0,C 180,E1 -6952.458,E2 -6952.458} C_VEL
LIN {X 0,Y 481.677,Z 260.299,A -85,B 0,C 180,E1 -6954.087,E2 -6954.087} C_VEL
LIN {X 0,Y 481.751,Z 260.293,A -85,B 0,C 180,E1 -6957.138,E2 -6957.138} C_VEL
LIN {X 0,Y 481.683,Z 260.296,A -85,B 0,C 180,E1 -6959.741,E2 -6959.741} C_VEL
LIN {X 0,Y 481.658,Z 260.295,A -85,B 0,C 180,E1 -6962.675,E2 -6962.675} C_VEL
LIN {X 0,Y 481.641,Z 260.299,A -85,B 0,C 180,E1 -6965.709,E2 -6965.709} C_VEL
LIN {X 0,Y 481.676,Z 260.296,A -85,B 0,C 180,E1 -6968.859,E2 -6968.859} C_VEL
LIN {X 0,Y 481.658,Z 260.299,A -85,B 0,C 180,E1 -6971.912,E2 -6971.912} C_VEL
LIN {X 0,Y 481.66,Z 260.294,A -85,B 0,C 180,E1 -6974.457,E2 -6974.457} C_VEL
LIN {X 0,Y 481.651,Z 260.301,A -85,B 0,C 180,E1 -6977.838,E2 -6977.838} C_VEL
LIN {X 0,Y 481.662,Z 260.293,A -85,B 0,C 180,E1 -6980.654,E2 -6980.654} C_VEL
LIN {X 0,Y 481.634,Z 260.304,A -85,B 0,C 180,E1 -6983.375,E2 -6983.375} C_VEL
LIN {X 0,Y 481.683,Z 260.293,A -85,B 0,C 180,E1 -6986.326,E2 -6986.326} C_VEL
LIN {X 0,Y 481.655,Z 260.298,A -85,B 0,C 180,E1 -6989.417,E2 -6989.417} C_VEL
LIN {X 0,Y 481.674,Z 260.295,A -85,B 0,C 180,E1 -6992.165,E2 -6992.165} C_VEL
LIN {X 0,Y 481.695,Z 260.29,A -85,B 0,C 180,E1 -6994.967,E2 -6994.967} C_VEL
LIN {X 0,Y 481.655,Z 260.301,A -85,B 0,C 180,E1 -6997.703,E2 -6997.703} C_VEL
LIN {X 0,Y 481.708,Z 260.29,A -85,B 0,C 180,E1 -7000.391,E2 -7000.391} C_VEL
LIN {X 0,Y 481.68,Z 260.29,A -85,B 0,C 180,E1 -7003.031,E2 -7003.031} C_VEL
LIN {X 0,Y 481.692,Z 260.293,A -85,B 0,C 180,E1 -7005.637,E2 -7005.637} C_VEL
LIN {X 0,Y 481.755,Z 260.282,A -85,B 0,C 180,E1 -7008.213,E2 -7008.213} C_VEL
LIN {X 0,Y 481.764,Z 260.283,A -85,B 0,C 180,E1 -7011.609,E2 -7011.609} C_VEL
LIN {X 0,Y 481.811,Z 260.277,A -85,B 0,C 180,E1 -7014.137,E2 -7014.137} C_VEL
LIN {X 0,Y 481.92,Z 260.262,A -85,B 0,C 180,E1 -7017.49,E2 -7017.49} C_VEL
LIN {X 0,Y 481.94,Z 260.262,A -85,B 0,C 180,E1 -7019.997,E2 -7019.997} C_VEL
LIN {X 0,Y 481.92,Z 260.265,A -85,B 0,C 180,E1 -7022.505,E2 -7022.505} C_VEL
LIN {X 0,Y 481.792,Z 260.277,A -85,B 0,C 180,E1 -7025.858,E2 -7025.858} C_VEL
LIN {X 0,Y 481.737,Z 260.29,A -85,B 0,C 180,E1 -7028.386,E2 -7028.386} C_VEL
LIN {X 0,Y 481.746,Z 260.284,A -85,B 0,C 180,E1 -7031.782,E2 -7031.782} C_VEL
LIN {X 0,Y 481.736,Z 260.283,A -85,B 0,C 180,E1 -7035.221,E2 -7035.221} C_VEL
LIN {X 0,Y 481.7,Z 260.293,A -85,B 0,C 180,E1 -7038.719,E2 -7038.719} C_VEL
LIN {X 0,Y 481.635,Z 260.297,A -85,B 0,C 180,E1 -7041.391,E2 -7041.391} C_VEL
LIN {X 0,Y 481.662,Z 260.299,A -85,B 0,C 180,E1 -7044.11,E2 -7044.11} C_VEL
LIN {X 0,Y 481.733,Z 260.287,A -85,B 0,C 180,E1 -7047.136,E2 -7047.136} C_VEL
LIN {X 0,Y 481.664,Z 260.295,A -85,B 0,C 180,E1 -7049.738,E2 -7049.738} C_VEL
LIN {X 0,Y 481.655,Z 260.303,A -85,B 0,C 180,E1 -7052.671,E2 -7052.671} C_VEL
LIN {X 0,Y 481.622,Z 260.295,A -85,B 0,C 180,E1 -7055.706,E2 -7055.706} C_VEL
LIN {X 0,Y 481.65,Z 260.301,A -85,B 0,C 180,E1 -7058.856,E2 -7058.856} C_VEL
LIN {X 0,Y 481.651,Z 260.299,A -85,B 0,C 180,E1 -7062.155,E2 -7062.155} C_VEL
LIN {X 0,Y 481.636,Z 260.302,A -85,B 0,C 180,E1 -7064.454,E2 -7064.454} C_VEL
LIN {X 0,Y 481.663,Z 260.3,A -85,B 0,C 180,E1 -7066.843,E2 -7066.843} C_VEL
LIN {X 0,Y 481.666,Z 260.297,A -85,B 0,C 180,E1 -7070.059,E2 -7070.059} C_VEL
LIN {X 0,Y 481.603,Z 260.308,A -85,B 0,C 180,E1 -7073.251,E2 -7073.251} C_VEL
LIN {X 0,Y 481.652,Z 260.389,A -85,B 0,C 180,E1 -7076.241,E2 -7076.241} C_VEL
LIN {X 0,Y 481.623,Z 270.658,A -85,B 0,C 180,E1 -7078.555,E2 -7078.555} C_VEL
LIN {X 0,Y 481.605,Z 277.228,A -85,B 0,C 180,E1 -7080.038,E2 -7080.038} C_VEL
LIN {X 0,Y 483.48,Z 287.728,A -85,B 0,C 180,E1 -7080.27,E2 -7080.27} C_VEL
LIN {X 0,Y 483.262,Z 329.559,A -85,B 0,C 180,E1 -7080.894,E2 -7080.894} C_VEL
LIN {X 0,Y 482.517,Z 335.429,A -85,B 0,C 180,E1 -7080.955,E2 -7080.955} C_VEL
LIN {X 0,Y 476.83,Z 353.419,A -85,B 0,C 180,E1 -7081.082,E2 -7081.082} C_VEL
LIN {X 0,Y 476.065,Z 359.169,A -85,B 0,C 180,E1 -7081.214,E2 -7081.214} C_VEL
LIN {X 0,Y 476.072,Z 360.09,A -85,B 0,C 180,E1 -7081.244,E2 -7081.244} C_VEL
LIN {X 0,Y 475.978,Z 369.026,A -85,B 0,C 180,E1 -7081.564,E2 -7081.564} C_VEL
LIN {X 0,Y 475.758,Z 377.748,A -85,B 0,C 180,E1 -7081.984,E2 -7081.984} C_VEL
LIN {X 0,Y 475.515,Z 386.754,A -85,B 0,C 180,E1 -7082.551,E2 -7082.551} C_VEL
LIN {X 0,Y 475.236,Z 394.852,A -85,B 0,C 180,E1 -7083.189,E2 -7083.189} C_VEL
LIN {X 0,Y 474.935,Z 402.045,A -85,B 0,C 180,E1 -7083.881,E2 -7083.881} C_VEL
LIN {X 0,Y 474.734,Z 408.065,A -85,B 0,C 180,E1 -7084.576,E2 -7084.576} C_VEL
LIN {X 0,Y 474.555,Z 413.195,A -85,B 0,C 180,E1 -7085.268,E2 -7085.268} C_VEL
LIN {X 0,Y 474.347,Z 418.885,A -85,B 0,C 180,E1 -7086.188,E2 -7086.188} C_VEL
LIN {X 0,Y 474.164,Z 423.261,A -85,B 0,C 180,E1 -7087.038,E2 -7087.038} C_VEL
LIN {X 0,Y 474.047,Z 426.536,A -85,B 0,C 180,E1 -7087.787,E2 -7087.787} C_VEL
LIN {X 0,Y 473.916,Z 430.865,A -85,B 0,C 180,E1 -7089.097,E2 -7089.097} C_VEL
LIN {X 0,Y 473.807,Z 433.213,A -85,B 0,C 180,E1 -7090.053,E2 -7090.053} C_VEL
LIN {X 0,Y 473.75,Z 434.826,A -85,B 0,C 180,E1 -7090.952,E2 -7090.952} C_VEL
LIN {X 0,Y 473.732,Z 435.824,A -85,B 0,C 180,E1 -7091.848,E2 -7091.848} C_VEL
LIN {X 0,Y 473.697,Z 436.22,A -85,B 0,C 180,E1 -7092.739,E2 -7092.739} C_VEL
LIN {X 0,Y 473.711,Z 436.096,A -85,B 0,C 180,E1 -7093.627,E2 -7093.627} C_VEL
LIN {X 0,Y 473.747,Z 435.343,A -85,B 0,C 180,E1 -7094.619,E2 -7094.619} C_VEL
LIN {X 0,Y 473.773,Z 434.322,A -85,B 0,C 180,E1 -7095.394,E2 -7095.394} C_VEL
LIN {X 0,Y 473.827,Z 432.629,A -85,B 0,C 180,E1 -7096.272,E2 -7096.272} C_VEL
LIN {X 0,Y 473.956,Z 428.88,A -85,B 0,C 180,E1 -7097.584,E2 -7097.584} C_VEL
LIN {X 0,Y 474.088,Z 423.723,A -85,B 0,C 180,E1 -7098.889,E2 -7098.889} C_VEL
LIN {X 0,Y 474.314,Z 418.163,A -85,B 0,C 180,E1 -7099.974,E2 -7099.974} C_VEL
LIN {X 0,Y 474.565,Z 411.196,A -85,B 0,C 180,E1 -7101.054,E2 -7101.054} C_VEL
LIN {X 0,Y 474.872,Z 403.175,A -85,B 0,C 180,E1 -7102.025,E2 -7102.025} C_VEL
LIN {X 0,Y 475.097,Z 395.863,A -85,B 0,C 180,E1 -7102.749,E2 -7102.749} C_VEL
LIN {X 0,Y 475.396,Z 387.506,A -85,B 0,C 180,E1 -7103.421,E2 -7103.421} C_VEL
LIN {X 0,Y 475.608,Z 379.221,A -85,B 0,C 180,E1 -7103.957,E2 -7103.957} C_VEL
LIN {X 0,Y 475.775,Z 370.808,A -85,B 0,C 180,E1 -7104.384,E2 -7104.384} C_VEL
LIN {X 0,Y 475.964,Z 361.614,A -85,B 0,C 180,E1 -7104.732,E2 -7104.732} C_VEL
LIN {X 0,Y 476.08,Z 353.431,A -85,B 0,C 180,E1 -7104.945,E2 -7104.945} C_VEL
LIN {X 0,Y 476.373,Z 288.042,A -85,B 0,C 180,E1 -7105.955,E2 -7105.955} C_VEL
LIN {X 0,Y 474.507,Z 277.6,A -85,B 0,C 180,E1 -7106.179,E2 -7106.179} C_VEL
LIN {X 0,Y 474.658,Z 265.013,A -85,B 0,C 180,E1 -7109.152,E2 -7109.152} C_VEL
LIN {X 0,Y 474.698,Z 261.166,A -85,B 0,C 180,E1 -7110.106,E2 -7110.106} C_VEL
LIN {X 0,Y 474.855,Z 261.144,A -85,B 0,C 180,E1 -7112.545,E2 -7112.545} C_VEL
LIN {X 0,Y 474.737,Z 261.159,A -85,B 0,C 180,E1 -7115.948,E2 -7115.948} C_VEL
LIN {X 0,Y 474.689,Z 261.164,A -85,B 0,C 180,E1 -7118.514,E2 -7118.514} C_VEL
LIN {X 0,Y 474.668,Z 261.167,A -85,B 0,C 180,E1 -7121.964,E2 -7121.964} C_VEL
LIN {X 0,Y 474.662,Z 261.174,A -85,B 0,C 180,E1 -7125.457,E2 -7125.457} C_VEL
LIN {X 0,Y 474.629,Z 261.174,A -85,B 0,C 180,E1 -7129.012,E2 -7129.012} C_VEL
LIN {X 0,Y 474.553,Z 261.184,A -85,B 0,C 180,E1 -7131.731,E2 -7131.731} C_VEL
LIN {X 0,Y 474.593,Z 261.175,A -85,B 0,C 180,E1 -7134.497,E2 -7134.497} C_VEL
LIN {X 0,Y 474.604,Z 261.18,A -85,B 0,C 180,E1 -7137.326,E2 -7137.326} C_VEL
LIN {X 0,Y 474.569,Z 261.179,A -85,B 0,C 180,E1 -7140.233,E2 -7140.233} C_VEL
LIN {X 0,Y 474.604,Z 261.178,A -85,B 0,C 180,E1 -7143.223,E2 -7143.223} C_VEL
LIN {X 0,Y 474.555,Z 261.18,A -85,B 0,C 180,E1 -7146.327,E2 -7146.327} C_VEL
LIN {X 0,Y 474.594,Z 261.183,A -85,B 0,C 180,E1 -7149.551,E2 -7149.551} C_VEL
LIN {X 0,Y 474.572,Z 261.179,A -85,B 0,C 180,E1 -7152.236,E2 -7152.236} C_VEL
LIN {X 0,Y 474.593,Z 261.179,A -85,B 0,C 180,E1 -7155.301,E2 -7155.301} C_VEL
LIN {X 0,Y 474.599,Z 261.177,A -85,B 0,C 180,E1 -7158.218,E2 -7158.218} C_VEL
LIN {X 0,Y 474.591,Z 261.182,A -85,B 0,C 180,E1 -7161.546,E2 -7161.546} C_VEL
LIN {X 0,Y 474.605,Z 261.174,A -85,B 0,C 180,E1 -7164.729,E2 -7164.729} C_VEL
LIN {X 0,Y 474.62,Z 261.181,A -85,B 0,C 180,E1 -7167.791,E2 -7167.791} C_VEL
LIN {X 0,Y 474.593,Z 261.176,A -85,B 0,C 180,E1 -7170.892,E2 -7170.892} C_VEL
LIN {X 0,Y 474.593,Z 261.181,A -85,B 0,C 180,E1 -7173.628,E2 -7173.628} C_VEL
LIN {X 0,Y 474.625,Z 261.172,A -85,B 0,C 180,E1 -7176.645,E2 -7176.645} C_VEL
LIN {X 0,Y 474.644,Z 261.175,A -85,B 0,C 180,E1 -7180.093,E2 -7180.093} C_VEL
LIN {X 0,Y 474.67,Z 261.262,A -85,B 0,C 180,E1 -7183.084,E2 -7183.084} C_VEL
LIN {X 0,Y 474.581,Z 270.981,A -85,B 0,C 180,E1 -7185.422,E2 -7185.422} C_VEL
LIN {X 0,Y 474.52,Z 277.421,A -85,B 0,C 180,E1 -7186.97,E2 -7186.97} C_VEL
LIN {X 0,Y 476.31,Z 288.634,A -85,B 0,C 180,E1 -7187.216,E2 -7187.216} C_VEL
LIN {X 0,Y 475.823,Z 354.62,A -85,B 0,C 180,E1 -7188.34,E2 -7188.34} C_VEL
LIN {X 0,Y 475.644,Z 364.386,A -85,B 0,C 180,E1 -7188.632,E2 -7188.632} C_VEL
LIN {X 0,Y 475.454,Z 373.75,A -85,B 0,C 180,E1 -7189.032,E2 -7189.032} C_VEL
LIN {X 0,Y 475.301,Z 383.196,A -85,B 0,C 180,E1 -7189.567,E2 -7189.567} C_VEL
LIN {X 0,Y 475.041,Z 393.358,A -85,B 0,C 180,E1 -7190.315,E2 -7190.315} C_VEL
LIN {X 0,Y 474.803,Z 401.292,A -85,B 0,C 180,E1 -7191.062,E2 -7191.062} C_VEL
LIN {X 0,Y 474.53,Z 408.717,A -85,B 0,C 180,E1 -7191.915,E2 -7191.915} C_VEL
LIN {X 0,Y 474.322,Z 414.848,A -85,B 0,C 180,E1 -7192.768,E2 -7192.768} C_VEL
LIN {X 0,Y 474.28,Z 420.082,A -85,B 0,C 180,E1 -7193.65,E2 -7193.65} C_VEL
LIN {X 0,Y 474.039,Z 424.163,A -85,B 0,C 180,E1 -7194.473,E2 -7194.473} C_VEL
LIN {X 0,Y 474.038,Z 427.651,A -85,B 0,C 180,E1 -7195.326,E2 -7195.326} C_VEL
LIN {X 0,Y 473.926,Z 431.649,A -85,B 0,C 180,E1 -7196.602,E2 -7196.602} C_VEL
LIN {X 0,Y 473.832,Z 433.567,A -85,B 0,C 180,E1 -7197.453,E2 -7197.453} C_VEL
LIN {X 0,Y 473.762,Z 434.955,A -85,B 0,C 180,E1 -7198.303,E2 -7198.303} C_VEL
LIN {X 0,Y 473.697,Z 435.839,A -85,B 0,C 180,E1 -7199.153,E2 -7199.153} C_VEL
LIN {X 0,Y 473.683,Z 436.18,A -85,B 0,C 180,E1 -7200.003,E2 -7200.003} C_VEL
LIN {X 0,Y 473.698,Z 435.94,A -85,B 0,C 180,E1 -7200.853,E2 -7200.853} C_VEL
LIN {X 0,Y 473.764,Z 435.197,A -85,B 0,C 180,E1 -7201.703,E2 -7201.703} C_VEL
LIN {X 0,Y 473.875,Z 433.949,A -85,B 0,C 180,E1 -7202.553,E2 -7202.553} C_VEL
LIN {X 0,Y 473.963,Z 431.054,A -85,B 0,C 180,E1 -7203.829,E2 -7203.829} C_VEL
LIN {X 0,Y 473.999,Z 426.872,A -85,B 0,C 180,E1 -7205.106,E2 -7205.106} C_VEL
LIN {X 0,Y 474.331,Z 420.977,A -85,B 0,C 180,E1 -7206.383,E2 -7206.383} C_VEL
LIN {X 0,Y 474.34,Z 416.366,A -85,B 0,C 180,E1 -7207.195,E2 -7207.195} C_VEL
LIN {X 0,Y 474.553,Z 410.181,A -85,B 0,C 180,E1 -7208.09,E2 -7208.09} C_VEL
LIN {X 0,Y 474.809,Z 403.004,A -85,B 0,C 180,E1 -7208.943,E2 -7208.943} C_VEL
LIN {X 0,Y 475.093,Z 394.179,A -85,B 0,C 180,E1 -7209.797,E2 -7209.797} C_VEL
LIN {X 0,Y 475.423,Z 384.193,A -85,B 0,C 180,E1 -7210.543,E2 -7210.543} C_VEL
LIN {X 0,Y 475.603,Z 373.824,A -85,B 0,C 180,E1 -7211.132,E2 -7211.132} C_VEL
LIN {X 0,Y 475.779,Z 363.63,A -85,B 0,C 180,E1 -7211.559,E2 -7211.559} C_VEL
LIN {X 0,Y 476.004,Z 350.439,A -85,B 0,C 180,E1 -7211.905,E2 -7211.905} C_VEL
LIN {X 0,Y 476.496,Z 288.151,A -85,B 0,C 180,E1 -7212.987,E2 -7212.987} C_VEL
LIN {X 0,Y 474.678,Z 278.436,A -85,B 0,C 180,E1 -7213.245,E2 -7213.245} C_VEL
LIN {X 0,Y 474.786,Z 265.12,A -85,B 0,C 180,E1 -7216.337,E2 -7216.337} C_VEL
LIN {X 0,Y 474.732,Z 261.168,A -85,B 0,C 180,E1 -7217.28,E2 -7217.28} C_VEL
LIN {X 0,Y 474.679,Z 261.17,A -85,B 0,C 180,E1 -7220.816,E2 -7220.816} C_VEL
LIN {X 0,Y 474.615,Z 261.176,A -85,B 0,C 180,E1 -7223.568,E2 -7223.568} C_VEL
LIN {X 0,Y 474.602,Z 261.182,A -85,B 0,C 180,E1 -7226.377,E2 -7226.377} C_VEL
LIN {X 0,Y 474.615,Z 261.175,A -85,B 0,C 180,E1 -7229.254,E2 -7229.254} C_VEL
LIN {X 0,Y 474.622,Z 261.18,A -85,B 0,C 180,E1 -7232.431,E2 -7232.431} C_VEL
LIN {X 0,Y 474.618,Z 261.174,A -85,B 0,C 180,E1 -7235.469,E2 -7235.469} C_VEL
LIN {X 0,Y 474.616,Z 261.181,A -85,B 0,C 180,E1 -7238.459,E2 -7238.459} C_VEL
LIN {X 0,Y 474.617,Z 261.174,A -85,B 0,C 180,E1 -7241.788,E2 -7241.788} C_VEL
LIN {X 0,Y 474.624,Z 261.178,A -85,B 0,C 180,E1 -7244.703,E2 -7244.703} C_VEL
LIN {X 0,Y 474.622,Z 261.175,A -85,B 0,C 180,E1 -7248.214,E2 -7248.214} C_VEL
LIN {X 0,Y 474.616,Z 261.173,A -85,B 0,C 180,E1 -7251.543,E2 -7251.543} C_VEL
LIN {X 0,Y 474.627,Z 261.179,A -85,B 0,C 180,E1 -7254.726,E2 -7254.726} C_VEL
LIN {X 0,Y 474.634,Z 261.172,A -85,B 0,C 180,E1 -7257.787,E2 -7257.787} C_VEL
LIN {X 0,Y 474.629,Z 261.176,A -85,B 0,C 180,E1 -7260.886,E2 -7260.886} C_VEL
LIN {X 0,Y 474.66,Z 261.17,A -85,B 0,C 180,E1 -7263.628,E2 -7263.628} C_VEL
LIN {X 0,Y 474.716,Z 261.358,A -85,B 0,C 180,E1 -7265.859,E2 -7265.859} C_VEL
LIN {X 0,Y 475.916,Z 269.152,A -85,B 0,C 180,E1 -7267.421,E2 -7267.421} C_VEL
LIN {X 0,Y 475.455,Z 284.469,A -85,B 0,C 180,E1 -7270.349,E2 -7270.349} C_VEL
LIN {X 0,Y 474.871,Z 302.058,A -85,B 0,C 180,E1 -7273.668,E2 -7273.668} C_VEL
LIN {X 0,Y 474.483,Z 318.641,A -85,B 0,C 180,E1 -7276.771,E2 -7276.771} C_VEL
LIN {X 0,Y 474.472,Z 319.353,A -85,B 0,C 180,E1 -7276.856,E2 -7276.856} C_VEL
LIN {X 0,Y 476.337,Z 336.515,A -85,B 0,C 180,E1 -7277.165,E2 -7277.165} C_VEL
LIN {X 0,Y 475.988,Z 396.775,A -85,B 0,C 180,E1 -7278.097,E2 -7278.097} C_VEL
LIN {X 0,Y 475.744,Z 406.515,A -85,B 0,C 180,E1 -7278.361,E2 -7278.361} C_VEL
LIN {X 0,Y 475.442,Z 417.607,A -85,B 0,C 180,E1 -7278.813,E2 -7278.813} C_VEL
LIN {X 0,Y 475.14,Z 428.458,A -85,B 0,C 180,E1 -7279.453,E2 -7279.453} C_VEL
LIN {X 0,Y 474.839,Z 436.887,A -85,B 0,C 180,E1 -7280.092,E2 -7280.092} C_VEL
LIN {X 0,Y 474.568,Z 444.852,A -85,B 0,C 180,E1 -7280.839,E2 -7280.839} C_VEL
LIN {X 0,Y 474.318,Z 452.292,A -85,B 0,C 180,E1 -7281.693,E2 -7281.693} C_VEL
LIN {X 0,Y 474.127,Z 459.84,A -85,B 0,C 180,E1 -7282.762,E2 -7282.762} C_VEL
LIN {X 0,Y 473.908,Z 466.739,A -85,B 0,C 180,E1 -7284.041,E2 -7284.041} C_VEL
LIN {X 0,Y 473.791,Z 471.961,A -85,B 0,C 180,E1 -7285.32,E2 -7285.32} C_VEL
LIN {X 0,Y 473.828,Z 474.639,A -85,B 0,C 180,E1 -7286.173,E2 -7286.173} C_VEL
LIN {X 0,Y 473.767,Z 477.566,A -85,B 0,C 180,E1 -7287.449,E2 -7287.449} C_VEL
LIN {X 0,Y 473.757,Z 478.833,A -85,B 0,C 180,E1 -7288.3,E2 -7288.3} C_VEL
LIN {X 0,Y 473.691,Z 479.621,A -85,B 0,C 180,E1 -7289.15,E2 -7289.15} C_VEL
LIN {X 0,Y 473.677,Z 479.916,A -85,B 0,C 180,E1 -7290,E2 -7290} C_VEL
LIN {X 0,Y 473.691,Z 479.618,A -85,B 0,C 180,E1 -7290.85,E2 -7290.85} C_VEL
LIN {X 0,Y 473.757,Z 478.837,A -85,B 0,C 180,E1 -7291.7,E2 -7291.7} C_VEL
LIN {X 0,Y 473.767,Z 477.577,A -85,B 0,C 180,E1 -7292.551,E2 -7292.551} C_VEL
LIN {X 0,Y 473.828,Z 474.657,A -85,B 0,C 180,E1 -7293.827,E2 -7293.827} C_VEL
LIN {X 0,Y 473.791,Z 471.997,A -85,B 0,C 180,E1 -7294.679,E2 -7294.679} C_VEL
LIN {X 0,Y 473.908,Z 466.795,A -85,B 0,C 180,E1 -7295.958,E2 -7295.958} C_VEL
LIN {X 0,Y 474.125,Z 459.958,A -85,B 0,C 180,E1 -7297.238,E2 -7297.238} C_VEL
LIN {X 0,Y 474.311,Z 452.485,A -85,B 0,C 180,E1 -7298.306,E2 -7298.306} C_VEL
LIN {X 0,Y 474.603,Z 445.127,A -85,B 0,C 180,E1 -7299.16,E2 -7299.16} C_VEL
LIN {X 0,Y 474.887,Z 437.258,A -85,B 0,C 180,E1 -7299.906,E2 -7299.906} C_VEL
LIN {X 0,Y 475.186,Z 428.959,A -85,B 0,C 180,E1 -7300.546,E2 -7300.546} C_VEL
LIN {X 0,Y 475.472,Z 418.403,A -85,B 0,C 180,E1 -7301.186,E2 -7301.186} C_VEL
LIN {X 0,Y 475.773,Z 407.073,A -85,B 0,C 180,E1 -7301.665,E2 -7301.665} C_VEL
LIN {X 0,Y 476.021,Z 397.762,A -85,B 0,C 180,E1 -7301.929,E2 -7301.929} C_VEL
LIN {X 0,Y 476.278,Z 370.495,A -85,B 0,C 180,E1 -7302.369,E2 -7302.369} C_VEL
LIN {X 0,Y 476.287,Z 333.893,A -85,B 0,C 180,E1 -7302.928,E2 -7302.928} C_VEL
LIN {X 0,Y 474.48,Z 318.805,A -85,B 0,C 180,E1 -7303.215,E2 -7303.215} C_VEL
LIN {X 0,Y 474.896,Z 302.12,A -85,B 0,C 180,E1 -7306.331,E2 -7306.331} C_VEL
LIN {X 0,Y 475.481,Z 284.549,A -85,B 0,C 180,E1 -7309.649,E2 -7309.649} C_VEL
LIN {X 0,Y 475.943,Z 269.276,A -85,B 0,C 180,E1 -7312.577,E2 -7312.577} C_VEL
LIN {X 0,Y 474.645,Z 261.175,A -85,B 0,C 180,E1 -7314.26,E2 -7314.26} C_VEL
LIN {X 0,Y 474.685,Z 261.171,A -85,B 0,C 180,E1 -7317.333,E2 -7317.333} C_VEL
LIN {X 0,Y 474.608,Z 261.177,A -85,B 0,C 180,E1 -7320.809,E2 -7320.809} C_VEL
LIN {X 0,Y 474.627,Z 261.175,A -85,B 0,C 180,E1 -7323.98,E2 -7323.98} C_VEL
LIN {X 0,Y 474.577,Z 261.178,A -85,B 0,C 180,E1 -7326.898,E2 -7326.898} C_VEL
LIN {X 0,Y 474.614,Z 261.179,A -85,B 0,C 180,E1 -7329.644,E2 -7329.644} C_VEL
LIN {X 0,Y 474.609,Z 261.175,A -85,B 0,C 180,E1 -7332.233,E2 -7332.233} C_VEL
LIN {X 0,Y 474.623,Z 261.176,A -85,B 0,C 180,E1 -7335.297,E2 -7335.297} C_VEL
LIN {X 0,Y 474.622,Z 261.173,A -85,B 0,C 180,E1 -7338.213,E2 -7338.213} C_VEL
LIN {X 0,Y 474.616,Z 261.177,A -85,B 0,C 180,E1 -7341.541,E2 -7341.541} C_VEL
LIN {X 0,Y 474.629,Z 261.168,A -85,B 0,C 180,E1 -7344.724,E2 -7344.724} C_VEL
LIN {X 0,Y 474.641,Z 261.174,A -85,B 0,C 180,E1 -7347.786,E2 -7347.786} C_VEL
LIN {X 0,Y 474.613,Z 261.173,A -85,B 0,C 180,E1 -7350.887,E2 -7350.887} C_VEL
LIN {X 0,Y 474.623,Z 261.175,A -85,B 0,C 180,E1 -7353.624,E2 -7353.624} C_VEL
LIN {X 0,Y 474.641,Z 261.169,A -85,B 0,C 180,E1 -7356.64,E2 -7356.64} C_VEL
LIN {X 0,Y 474.658,Z 261.172,A -85,B 0,C 180,E1 -7360.088,E2 -7360.088} C_VEL
LIN {X 0,Y 474.64,Z 261.167,A -85,B 0,C 180,E1 -7362.772,E2 -7362.772} C_VEL
LIN {X 0,Y 474.651,Z 261.168,A -85,B 0,C 180,E1 -7365.419,E2 -7365.419} C_VEL
LIN {X 0,Y 474.708,Z 261.162,A -85,B 0,C 180,E1 -7368.035,E2 -7368.035} C_VEL
LIN {X 0,Y 474.729,Z 261.158,A -85,B 0,C 180,E1 -7371.484,E2 -7371.484} C_VEL
LIN {X 0,Y 474.774,Z 261.154,A -85,B 0,C 180,E1 -7374.05,E2 -7374.05} C_VEL
LIN {X 0,Y 474.885,Z 261.138,A -85,B 0,C 180,E1 -7377.453,E2 -7377.453} C_VEL
LIN {X 0,Y 474.91,Z 261.137,A -85,B 0,C 180,E1 -7379.997,E2 -7379.997} C_VEL
LIN {X 0,Y 474.885,Z 261.141,A -85,B 0,C 180,E1 -7382.542,E2 -7382.542} C_VEL
LIN {X 0,Y 474.753,Z 261.155,A -85,B 0,C 180,E1 -7385.945,E2 -7385.945} C_VEL
LIN {X 0,Y 474.709,Z 261.164,A -85,B 0,C 180,E1 -7388.511,E2 -7388.511} C_VEL
LIN {X 0,Y 474.699,Z 261.164,A -85,B 0,C 180,E1 -7391.959,E2 -7391.959} C_VEL
LIN {X 0,Y 474.693,Z 261.16,A -85,B 0,C 180,E1 -7395.452,E2 -7395.452} C_VEL
LIN {X 0,Y 474.654,Z 261.168,A -85,B 0,C 180,E1 -7399.007,E2 -7399.007} C_VEL
LIN {X 0,Y 474.578,Z 261.177,A -85,B 0,C 180,E1 -7401.726,E2 -7401.726} C_VEL
LIN {X 0,Y 474.645,Z 261.174,A -85,B 0,C 180,E1 -7404.49,E2 -7404.49} C_VEL
LIN {X 0,Y 474.667,Z 261.166,A -85,B 0,C 180,E1 -7407.331,E2 -7407.331} C_VEL
LIN {X 0,Y 474.59,Z 261.181,A -85,B 0,C 180,E1 -7410.227,E2 -7410.227} C_VEL
LIN {X 0,Y 474.625,Z 261.173,A -85,B 0,C 180,E1 -7413.217,E2 -7413.217} C_VEL
LIN {X 0,Y 474.572,Z 261.177,A -85,B 0,C 180,E1 -7416.32,E2 -7416.32} C_VEL
LIN {X 0,Y 474.606,Z 261.173,A -85,B 0,C 180,E1 -7419.644,E2 -7419.644} C_VEL
LIN {X 0,Y 474.629,Z 261.175,A -85,B 0,C 180,E1 -7422.927,E2 -7422.927} C_VEL
LIN {X 0,Y 474.593,Z 261.177,A -85,B 0,C 180,E1 -7425.893,E2 -7425.893} C_VEL
LIN {X 0,Y 474.62,Z 261.177,A -85,B 0,C 180,E1 -7429.035,E2 -7429.035} C_VEL
LIN {X 0,Y 474.592,Z 261.179,A -85,B 0,C 180,E1 -7431.7,E2 -7431.7} C_VEL
LIN {X 0,Y 474.603,Z 261.183,A -85,B 0,C 180,E1 -7434.724,E2 -7434.724} C_VEL
LIN {X 0,Y 474.619,Z 261.348,A -85,B 0,C 180,E1 -7436.148,E2 -7436.148} C_VEL
LIN {X 0,Y 474.631,Z 271.834,A -85,B 0,C 180,E1 -7438.537,E2 -7438.537} C_VEL
LIN {X 0,Y 474.598,Z 277.547,A -85,B 0,C 180,E1 -7439.836,E2 -7439.836} C_VEL
LIN {X 0,Y 476.612,Z 288.785,A -85,B 0,C 180,E1 -7440.082,E2 -7440.082} C_VEL
LIN {X 0,Y 476.165,Z 354.049,A -85,B 0,C 180,E1 -7441.094,E2 -7441.094} C_VEL
LIN {X 0,Y 476.072,Z 360.09,A -85,B 0,C 180,E1 -7441.244,E2 -7441.244} C_VEL
LIN {X 0,Y 475.43,Z 365.921,A -85,B 0,C 180,E1 -7441.417,E2 -7441.417} C_VEL
LIN {X 0,Y 472.555,Z 375.281,A -85,B 0,C 180,E1 -7441.753,E2 -7441.753} C_VEL
LIN {X 0,Y 469.413,Z 383.815,A -85,B 0,C 180,E1 -7442.165,E2 -7442.165} C_VEL
LIN {X 0,Y 468.523,Z 388.76,A -85,B 0,C 180,E1 -7442.501,E2 -7442.501} C_VEL
LIN {X 0,Y 468.142,Z 398.795,A -85,B 0,C 180,E1 -7443.353,E2 -7443.353} C_VEL
LIN {X 0,Y 467.755,Z 407.685,A -85,B 0,C 180,E1 -7444.345,E2 -7444.345} C_VEL
LIN {X 0,Y 467.537,Z 413.333,A -85,B 0,C 180,E1 -7445.109,E2 -7445.109} C_VEL
LIN {X 0,Y 467.317,Z 419.058,A -85,B 0,C 180,E1 -7446.043,E2 -7446.043} C_VEL
LIN {X 0,Y 467.111,Z 423.75,A -85,B 0,C 180,E1 -7446.972,E2 -7446.972} C_VEL
LIN {X 0,Y 466.9,Z 429.184,A -85,B 0,C 180,E1 -7448.359,E2 -7448.359} C_VEL
LIN {X 0,Y 466.787,Z 433.047,A -85,B 0,C 180,E1 -7449.74,E2 -7449.74} C_VEL
LIN {X 0,Y 466.674,Z 434.758,A -85,B 0,C 180,E1 -7450.652,E2 -7450.652} C_VEL
LIN {X 0,Y 466.642,Z 435.89,A -85,B 0,C 180,E1 -7451.577,E2 -7451.577} C_VEL
LIN {X 0,Y 466.611,Z 436.456,A -85,B 0,C 180,E1 -7452.468,E2 -7452.468} C_VEL
LIN {X 0,Y 466.621,Z 436.518,A -85,B 0,C 180,E1 -7453.371,E2 -7453.371} C_VEL
LIN {X 0,Y 466.676,Z 435.789,A -85,B 0,C 180,E1 -7454.523,E2 -7454.523} C_VEL
LIN {X 0,Y 466.67,Z 435.064,A -85,B 0,C 180,E1 -7455.166,E2 -7455.166} C_VEL
LIN {X 0,Y 466.775,Z 432.457,A -85,B 0,C 180,E1 -7456.504,E2 -7456.504} C_VEL
LIN {X 0,Y 466.867,Z 430.054,A -85,B 0,C 180,E1 -7457.392,E2 -7457.392} C_VEL
LIN {X 0,Y 466.99,Z 425.132,A -85,B 0,C 180,E1 -7458.718,E2 -7458.718} C_VEL
LIN {X 0,Y 467.175,Z 421.002,A -85,B 0,C 180,E1 -7459.6,E2 -7459.6} C_VEL
LIN {X 0,Y 467.321,Z 416.042,A -85,B 0,C 180,E1 -7460.478,E2 -7460.478} C_VEL
LIN {X 0,Y 467.56,Z 410.036,A -85,B 0,C 180,E1 -7461.355,E2 -7461.355} C_VEL
LIN {X 0,Y 467.914,Z 402.699,A -85,B 0,C 180,E1 -7462.231,E2 -7462.231} C_VEL
LIN {X 0,Y 468.124,Z 395.351,A -85,B 0,C 180,E1 -7462.955,E2 -7462.955} C_VEL
LIN {X 0,Y 468.406,Z 388.174,A -85,B 0,C 180,E1 -7463.539,E2 -7463.539} C_VEL
LIN {X 0,Y 468.629,Z 379.974,A -85,B 0,C 180,E1 -7464.082,E2 -7464.082} C_VEL
LIN {X 0,Y 468.813,Z 371.681,A -85,B 0,C 180,E1 -7464.516,E2 -7464.516} C_VEL
LIN {X 0,Y 469.009,Z 362.694,A -85,B 0,C 180,E1 -7464.869,E2 -7464.869} C_VEL
LIN {X 0,Y 469.123,Z 353.677,A -85,B 0,C 180,E1 -7465.112,E2 -7465.112} C_VEL
LIN {X 0,Y 469.384,Z 288.362,A -85,B 0,C 180,E1 -7466.137,E2 -7466.137} C_VEL
LIN {X 0,Y 467.473,Z 277.878,A -85,B 0,C 180,E1 -7466.364,E2 -7466.364} C_VEL
LIN {X 0,Y 467.728,Z 264.369,A -85,B 0,C 180,E1 -7469.57,E2 -7469.57} C_VEL
LIN {X 0,Y 467.666,Z 262.043,A -85,B 0,C 180,E1 -7470.162,E2 -7470.162} C_VEL
LIN {X 0,Y 467.821,Z 262.02,A -85,B 0,C 180,E1 -7472.583,E2 -7472.583} C_VEL
LIN {X 0,Y 467.701,Z 262.035,A -85,B 0,C 180,E1 -7476.038,E2 -7476.038} C_VEL
LIN {X 0,Y 467.643,Z 262.042,A -85,B 0,C 180,E1 -7478.644,E2 -7478.644} C_VEL
LIN {X 0,Y 467.619,Z 262.044,A -85,B 0,C 180,E1 -7482.147,E2 -7482.147} C_VEL
LIN {X 0,Y 467.602,Z 262.05,A -85,B 0,C 180,E1 -7485.696,E2 -7485.696} C_VEL
LIN {X 0,Y 467.581,Z 262.05,A -85,B 0,C 180,E1 -7488.766,E2 -7488.766} C_VEL
LIN {X 0,Y 467.545,Z 262.06,A -85,B 0,C 180,E1 -7491.27,E2 -7491.27} C_VEL
LIN {X 0,Y 467.521,Z 262.058,A -85,B 0,C 180,E1 -7493.946,E2 -7493.946} C_VEL
LIN {X 0,Y 467.529,Z 262.056,A -85,B 0,C 180,E1 -7496.806,E2 -7496.806} C_VEL
LIN {X 0,Y 467.514,Z 262.062,A -85,B 0,C 180,E1 -7499.741,E2 -7499.741} C_VEL
LIN {X 0,Y 467.551,Z 262.053,A -85,B 0,C 180,E1 -7502.761,E2 -7502.761} C_VEL
LIN {X 0,Y 467.522,Z 262.06,A -85,B 0,C 180,E1 -7505.893,E2 -7505.893} C_VEL
LIN {X 0,Y 467.524,Z 262.059,A -85,B 0,C 180,E1 -7509.151,E2 -7509.151} C_VEL
LIN {X 0,Y 467.541,Z 262.059,A -85,B 0,C 180,E1 -7511.407,E2 -7511.407} C_VEL
LIN {X 0,Y 467.542,Z 262.055,A -85,B 0,C 180,E1 -7514.951,E2 -7514.951} C_VEL
LIN {X 0,Y 467.568,Z 262.056,A -85,B 0,C 180,E1 -7517.443,E2 -7517.443} C_VEL
LIN {X 0,Y 467.54,Z 262.055,A -85,B 0,C 180,E1 -7520.856,E2 -7520.856} C_VEL
LIN {X 0,Y 467.541,Z 262.056,A -85,B 0,C 180,E1 -7524.265,E2 -7524.265} C_VEL
LIN {X 0,Y 467.564,Z 262.054,A -85,B 0,C 180,E1 -7527.325,E2 -7527.325} C_VEL
LIN {X 0,Y 467.543,Z 262.054,A -85,B 0,C 180,E1 -7530.674,E2 -7530.674} C_VEL
LIN {X 0,Y 467.546,Z 262.055,A -85,B 0,C 180,E1 -7533.2,E2 -7533.2} C_VEL
LIN {X 0,Y 467.58,Z 262.051,A -85,B 0,C 180,E1 -7536.473,E2 -7536.473} C_VEL
LIN {X 0,Y 467.613,Z 262.051,A -85,B 0,C 180,E1 -7539.781,E2 -7539.781} C_VEL
LIN {X 0,Y 467.604,Z 262.131,A -85,B 0,C 180,E1 -7543.045,E2 -7543.045} C_VEL
LIN {X 0,Y 467.518,Z 272.864,A -85,B 0,C 180,E1 -7545.642,E2 -7545.642} C_VEL
LIN {X 0,Y 467.515,Z 277.893,A -85,B 0,C 180,E1 -7546.81,E2 -7546.81} C_VEL
LIN {X 0,Y 469.358,Z 288.88,A -85,B 0,C 180,E1 -7547.049,E2 -7547.049} C_VEL
LIN {X 0,Y 468.834,Z 354.435,A -85,B 0,C 180,E1 -7548.191,E2 -7548.191} C_VEL
LIN {X 0,Y 468.632,Z 365.025,A -85,B 0,C 180,E1 -7548.514,E2 -7548.514} C_VEL
LIN {X 0,Y 468.432,Z 374.299,A -85,B 0,C 180,E1 -7548.92,E2 -7548.92} C_VEL
LIN {X 0,Y 468.255,Z 384.568,A -85,B 0,C 180,E1 -7549.518,E2 -7549.518} C_VEL
LIN {X 0,Y 467.992,Z 394.393,A -85,B 0,C 180,E1 -7550.277,E2 -7550.277} C_VEL
LIN {X 0,Y 467.685,Z 403.211,A -85,B 0,C 180,E1 -7551.143,E2 -7551.143} C_VEL
LIN {X 0,Y 467.424,Z 410.389,A -85,B 0,C 180,E1 -7552.009,E2 -7552.009} C_VEL
LIN {X 0,Y 467.282,Z 417.683,A -85,B 0,C 180,E1 -7553.092,E2 -7553.092} C_VEL
LIN {X 0,Y 467.115,Z 422.36,A -85,B 0,C 180,E1 -7553.957,E2 -7553.957} C_VEL
LIN {X 0,Y 466.959,Z 427.852,A -85,B 0,C 180,E1 -7555.255,E2 -7555.255} C_VEL
LIN {X 0,Y 466.858,Z 431.884,A -85,B 0,C 180,E1 -7556.551,E2 -7556.551} C_VEL
LIN {X 0,Y 466.75,Z 433.831,A -85,B 0,C 180,E1 -7557.414,E2 -7557.414} C_VEL
LIN {X 0,Y 466.698,Z 435.243,A -85,B 0,C 180,E1 -7558.277,E2 -7558.277} C_VEL
LIN {X 0,Y 466.627,Z 436.147,A -85,B 0,C 180,E1 -7559.14,E2 -7559.14} C_VEL
LIN {X 0,Y 466.611,Z 436.497,A -85,B 0,C 180,E1 -7560.003,E2 -7560.003} C_VEL
LIN {X 0,Y 466.628,Z 436.271,A -85,B 0,C 180,E1 -7560.866,E2 -7560.866} C_VEL
LIN {X 0,Y 466.701,Z 435.542,A -85,B 0,C 180,E1 -7561.729,E2 -7561.729} C_VEL
LIN {X 0,Y 466.789,Z 434.308,A -85,B 0,C 180,E1 -7562.592,E2 -7562.592} C_VEL
LIN {X 0,Y 466.901,Z 431.418,A -85,B 0,C 180,E1 -7563.887,E2 -7563.887} C_VEL
LIN {X 0,Y 467,Z 428.735,A -85,B 0,C 180,E1 -7564.75,E2 -7564.75} C_VEL
LIN {X 0,Y 466.992,Z 425.417,A -85,B 0,C 180,E1 -7565.616,E2 -7565.616} C_VEL
LIN {X 0,Y 467.299,Z 420.338,A -85,B 0,C 180,E1 -7566.671,E2 -7566.671} C_VEL
LIN {X 0,Y 467.372,Z 415.221,A -85,B 0,C 180,E1 -7567.541,E2 -7567.541} C_VEL
LIN {X 0,Y 467.603,Z 408.903,A -85,B 0,C 180,E1 -7568.429,E2 -7568.429} C_VEL
LIN {X 0,Y 467.947,Z 400.376,A -85,B 0,C 180,E1 -7569.403,E2 -7569.403} C_VEL
LIN {X 0,Y 468.29,Z 390.5,A -85,B 0,C 180,E1 -7570.268,E2 -7570.268} C_VEL
LIN {X 0,Y 468.489,Z 382.863,A -85,B 0,C 180,E1 -7570.81,E2 -7570.81} C_VEL
LIN {X 0,Y 468.686,Z 373.203,A -85,B 0,C 180,E1 -7571.353,E2 -7571.353} C_VEL
LIN {X 0,Y 468.904,Z 361.985,A -85,B 0,C 180,E1 -7571.813,E2 -7571.813} C_VEL
LIN {X 0,Y 469.088,Z 349.957,A -85,B 0,C 180,E1 -7572.11,E2 -7572.11} C_VEL
LIN {X 0,Y 469.603,Z 288.736,A -85,B 0,C 180,E1 -7573.208,E2 -7573.208} C_VEL
LIN {X 0,Y 467.656,Z 278.717,A -85,B 0,C 180,E1 -7573.473,E2 -7573.473} C_VEL
LIN {X 0,Y 467.798,Z 267.199,A -85,B 0,C 180,E1 -7576.185,E2 -7576.185} C_VEL
LIN {X 0,Y 467.676,Z 262.048,A -85,B 0,C 180,E1 -7577.408,E2 -7577.408} C_VEL
LIN {X 0,Y 467.63,Z 262.052,A -85,B 0,C 180,E1 -7580.225,E2 -7580.225} C_VEL
LIN {X 0,Y 467.564,Z 262.057,A -85,B 0,C 180,E1 -7583.946,E2 -7583.946} C_VEL
LIN {X 0,Y 467.561,Z 262.057,A -85,B 0,C 180,E1 -7586.806,E2 -7586.806} C_VEL
LIN {X 0,Y 467.555,Z 262.055,A -85,B 0,C 180,E1 -7589.74,E2 -7589.74} C_VEL
LIN {X 0,Y 467.587,Z 262.054,A -85,B 0,C 180,E1 -7592.76,E2 -7592.76} C_VEL
LIN {X 0,Y 467.559,Z 262.055,A -85,B 0,C 180,E1 -7595.891,E2 -7595.891} C_VEL
LIN {X 0,Y 467.56,Z 262.054,A -85,B 0,C 180,E1 -7599.149,E2 -7599.149} C_VEL
LIN {X 0,Y 467.575,Z 262.051,A -85,B 0,C 180,E1 -7601.405,E2 -7601.405} C_VEL
LIN {X 0,Y 467.574,Z 262.053,A -85,B 0,C 180,E1 -7604.948,E2 -7604.948} C_VEL
LIN {X 0,Y 467.581,Z 262.055,A -85,B 0,C 180,E1 -7608.597,E2 -7608.597} C_VEL
LIN {X 0,Y 467.569,Z 262.052,A -85,B 0,C 180,E1 -7611.956,E2 -7611.956} C_VEL
LIN {X 0,Y 467.563,Z 262.054,A -85,B 0,C 180,E1 -7615.167,E2 -7615.167} C_VEL
LIN {X 0,Y 467.585,Z 262.053,A -85,B 0,C 180,E1 -7618.26,E2 -7618.26} C_VEL
LIN {X 0,Y 467.581,Z 262.053,A -85,B 0,C 180,E1 -7621.251,E2 -7621.251} C_VEL
LIN {X 0,Y 467.604,Z 262.05,A -85,B 0,C 180,E1 -7624.159,E2 -7624.159} C_VEL
LIN {X 0,Y 467.62,Z 262.079,A -85,B 0,C 180,E1 -7625.705,E2 -7625.705} C_VEL
LIN {X 0,Y 468.895,Z 269.881,A -85,B 0,C 180,E1 -7627.297,E2 -7627.297} C_VEL
LIN {X 0,Y 468.484,Z 282.872,A -85,B 0,C 180,E1 -7629.816,E2 -7629.816} C_VEL
LIN {X 0,Y 467.895,Z 299.306,A -85,B 0,C 180,E1 -7632.968,E2 -7632.968} C_VEL
LIN {X 0,Y 467.482,Z 315.673,A -85,B 0,C 180,E1 -7636.081,E2 -7636.081} C_VEL
LIN {X 0,Y 467.436,Z 318.873,A -85,B 0,C 180,E1 -7636.667,E2 -7636.667} C_VEL
LIN {X 0,Y 469.381,Z 337.029,A -85,B 0,C 180,E1 -7636.999,E2 -7636.999} C_VEL
LIN {X 0,Y 469.04,Z 395.806,A -85,B 0,C 180,E1 -7637.918,E2 -7637.918} C_VEL
LIN {X 0,Y 468.802,Z 404.943,A -85,B 0,C 180,E1 -7638.159,E2 -7638.159} C_VEL
LIN {X 0,Y 468.512,Z 414.58,A -85,B 0,C 180,E1 -7638.535,E2 -7638.535} C_VEL
LIN {X 0,Y 468.226,Z 424.684,A -85,B 0,C 180,E1 -7639.076,E2 -7639.076} C_VEL
LIN {X 0,Y 467.88,Z 435.173,A -85,B 0,C 180,E1 -7639.834,E2 -7639.834} C_VEL
LIN {X 0,Y 467.591,Z 443.374,A -85,B 0,C 180,E1 -7640.592,E2 -7640.592} C_VEL
LIN {X 0,Y 467.345,Z 450.146,A -85,B 0,C 180,E1 -7641.351,E2 -7641.351} C_VEL
LIN {X 0,Y 467.088,Z 456.565,A -85,B 0,C 180,E1 -7642.217,E2 -7642.217} C_VEL
LIN {X 0,Y 466.997,Z 461.906,A -85,B 0,C 180,E1 -7643.085,E2 -7643.085} C_VEL
LIN {X 0,Y 466.818,Z 466.354,A -85,B 0,C 180,E1 -7643.95,E2 -7643.95} C_VEL
LIN {X 0,Y 466.799,Z 470.062,A -85,B 0,C 180,E1 -7644.817,E2 -7644.817} C_VEL
LIN {X 0,Y 466.669,Z 473.087,A -85,B 0,C 180,E1 -7645.681,E2 -7645.681} C_VEL
LIN {X 0,Y 466.758,Z 475.441,A -85,B 0,C 180,E1 -7646.547,E2 -7646.547} C_VEL
LIN {X 0,Y 466.687,Z 477.217,A -85,B 0,C 180,E1 -7647.41,E2 -7647.41} C_VEL
LIN {X 0,Y 466.662,Z 478.494,A -85,B 0,C 180,E1 -7648.274,E2 -7648.274} C_VEL
LIN {X 0,Y 466.623,Z 479.291,A -85,B 0,C 180,E1 -7649.137,E2 -7649.137} C_VEL
LIN {X 0,Y 466.606,Z 479.589,A -85,B 0,C 180,E1 -7650,E2 -7650} C_VEL
LIN {X 0,Y 466.623,Z 479.296,A -85,B 0,C 180,E1 -7650.863,E2 -7650.863} C_VEL
LIN {X 0,Y 466.662,Z 478.522,A -85,B 0,C 180,E1 -7651.726,E2 -7651.726} C_VEL
LIN {X 0,Y 466.687,Z 477.272,A -85,B 0,C 180,E1 -7652.589,E2 -7652.589} C_VEL
LIN {X 0,Y 466.758,Z 475.525,A -85,B 0,C 180,E1 -7653.453,E2 -7653.453} C_VEL
LIN {X 0,Y 466.718,Z 471.71,A -85,B 0,C 180,E1 -7654.751,E2 -7654.751} C_VEL
LIN {X 0,Y 466.82,Z 466.516,A -85,B 0,C 180,E1 -7656.049,E2 -7656.049} C_VEL
LIN {X 0,Y 467.052,Z 459.699,A -85,B 0,C 180,E1 -7657.348,E2 -7657.348} C_VEL
LIN {X 0,Y 467.276,Z 452.246,A -85,B 0,C 180,E1 -7658.432,E2 -7658.432} C_VEL
LIN {X 0,Y 467.553,Z 444.904,A -85,B 0,C 180,E1 -7659.299,E2 -7659.299} C_VEL
LIN {X 0,Y 467.876,Z 437.058,A -85,B 0,C 180,E1 -7660.056,E2 -7660.056} C_VEL
LIN {X 0,Y 468.202,Z 428.788,A -85,B 0,C 180,E1 -7660.705,E2 -7660.705} C_VEL
LIN {X 0,Y 468.509,Z 418.282,A -85,B 0,C 180,E1 -7661.355,E2 -7661.355} C_VEL
LIN {X 0,Y 468.839,Z 407.101,A -85,B 0,C 180,E1 -7661.84,E2 -7661.84} C_VEL
LIN {X 0,Y 469.147,Z 397.09,A -85,B 0,C 180,E1 -7662.125,E2 -7662.125} C_VEL
LIN {X 0,Y 469.377,Z 362.614,A -85,B 0,C 180,E1 -7662.684,E2 -7662.684} C_VEL
LIN {X 0,Y 469.355,Z 334.151,A -85,B 0,C 180,E1 -7663.128,E2 -7663.128} C_VEL
LIN {X 0,Y 467.432,Z 318.387,A -85,B 0,C 180,E1 -7663.448,E2 -7663.448} C_VEL
LIN {X 0,Y 467.86,Z 302.913,A -85,B 0,C 180,E1 -7666.386,E2 -7666.386} C_VEL
LIN {X 0,Y 468.492,Z 285.483,A -85,B 0,C 180,E1 -7669.726,E2 -7669.726} C_VEL
LIN {X 0,Y 468.962,Z 271.42,A -85,B 0,C 180,E1 -7672.467,E2 -7672.467} C_VEL
LIN {X 0,Y 468.579,Z 267.218,A -85,B 0,C 180,E1 -7673.318,E2 -7673.318} C_VEL
LIN {X 0,Y 467.611,Z 262.052,A -85,B 0,C 180,E1 -7674.413,E2 -7674.413} C_VEL
LIN {X 0,Y 467.625,Z 262.048,A -85,B 0,C 180,E1 -7677.769,E2 -7677.769} C_VEL
LIN {X 0,Y 467.572,Z 262.056,A -85,B 0,C 180,E1 -7681.044,E2 -7681.044} C_VEL
LIN {X 0,Y 467.582,Z 262.051,A -85,B 0,C 180,E1 -7684.239,E2 -7684.239} C_VEL
LIN {X 0,Y 467.553,Z 262.056,A -85,B 0,C 180,E1 -7687.185,E2 -7687.185} C_VEL
LIN {X 0,Y 467.578,Z 262.05,A -85,B 0,C 180,E1 -7690.264,E2 -7690.264} C_VEL
LIN {X 0,Y 467.567,Z 262.052,A -85,B 0,C 180,E1 -7692.562,E2 -7692.562} C_VEL
LIN {X 0,Y 467.572,Z 262.051,A -85,B 0,C 180,E1 -7695.051,E2 -7695.051} C_VEL
LIN {X 0,Y 467.58,Z 262.049,A -85,B 0,C 180,E1 -7698.596,E2 -7698.596} C_VEL
LIN {X 0,Y 467.57,Z 262.054,A -85,B 0,C 180,E1 -7701.954,E2 -7701.954} C_VEL
LIN {X 0,Y 467.564,Z 262.051,A -85,B 0,C 180,E1 -7705.165,E2 -7705.165} C_VEL
LIN {X 0,Y 467.588,Z 262.047,A -85,B 0,C 180,E1 -7708.258,E2 -7708.258} C_VEL
LIN {X 0,Y 467.561,Z 262.054,A -85,B 0,C 180,E1 -7711.247,E2 -7711.247} C_VEL
LIN {X 0,Y 467.591,Z 262.05,A -85,B 0,C 180,E1 -7714.157,E2 -7714.157} C_VEL
LIN {X 0,Y 467.582,Z 262.049,A -85,B 0,C 180,E1 -7716.994,E2 -7716.994} C_VEL
LIN {X 0,Y 467.627,Z 262.047,A -85,B 0,C 180,E1 -7719.775,E2 -7719.775} C_VEL
LIN {X 0,Y 467.601,Z 262.045,A -85,B 0,C 180,E1 -7722.504,E2 -7722.504} C_VEL
LIN {X 0,Y 467.61,Z 262.043,A -85,B 0,C 180,E1 -7725.194,E2 -7725.194} C_VEL
LIN {X 0,Y 467.66,Z 262.043,A -85,B 0,C 180,E1 -7727.852,E2 -7727.852} C_VEL
LIN {X 0,Y 467.683,Z 262.035,A -85,B 0,C 180,E1 -7731.355,E2 -7731.355} C_VEL
LIN {X 0,Y 467.738,Z 262.03,A -85,B 0,C 180,E1 -7733.96,E2 -7733.96} C_VEL
LIN {X 0,Y 467.85,Z 262.015,A -85,B 0,C 180,E1 -7737.414,E2 -7737.414} C_VEL
LIN {X 0,Y 467.88,Z 262.012,A -85,B 0,C 180,E1 -7739.997,E2 -7739.997} C_VEL
LIN {X 0,Y 467.85,Z 262.017,A -85,B 0,C 180,E1 -7742.58,E2 -7742.58} C_VEL
LIN {X 0,Y 467.715,Z 262.032,A -85,B 0,C 180,E1 -7746.035,E2 -7746.035} C_VEL
LIN {X 0,Y 467.667,Z 262.04,A -85,B 0,C 180,E1 -7748.64,E2 -7748.64} C_VEL
LIN {X 0,Y 467.651,Z 262.044,A -85,B 0,C 180,E1 -7752.142,E2 -7752.142} C_VEL
LIN {X 0,Y 467.632,Z 262.041,A -85,B 0,C 180,E1 -7755.692,E2 -7755.692} C_VEL
LIN {X 0,Y 467.613,Z 262.044,A -85,B 0,C 180,E1 -7759.305,E2 -7759.305} C_VEL
LIN {X 0,Y 467.524,Z 262.059,A -85,B 0,C 180,E1 -7762.071,E2 -7762.071} C_VEL
LIN {X 0,Y 467.59,Z 262.05,A -85,B 0,C 180,E1 -7764.884,E2 -7764.884} C_VEL
LIN {X 0,Y 467.606,Z 262.046,A -85,B 0,C 180,E1 -7767.766,E2 -7767.766} C_VEL
LIN {X 0,Y 467.552,Z 262.053,A -85,B 0,C 180,E1 -7771.042,E2 -7771.042} C_VEL
LIN {X 0,Y 467.572,Z 262.055,A -85,B 0,C 180,E1 -7774.239,E2 -7774.239} C_VEL
LIN {X 0,Y 467.53,Z 262.057,A -85,B 0,C 180,E1 -7777.183,E2 -7777.183} C_VEL
LIN {X 0,Y 467.557,Z 262.055,A -85,B 0,C 180,E1 -7780.261,E2 -7780.261} C_VEL
LIN {X 0,Y 467.596,Z 262.056,A -85,B 0,C 180,E1 -7782.568,E2 -7782.568} C_VEL
LIN {X 0,Y 467.549,Z 262.057,A -85,B 0,C 180,E1 -7786.174,E2 -7786.174} C_VEL
LIN {X 0,Y 467.564,Z 262.058,A -85,B 0,C 180,E1 -7788.719,E2 -7788.719} C_VEL
LIN {X 0,Y 467.55,Z 262.058,A -85,B 0,C 180,E1 -7791.404,E2 -7791.404} C_VEL
LIN {X 0,Y 467.535,Z 262.06,A -85,B 0,C 180,E1 -7794.258,E2 -7794.258} C_VEL
LIN {X 0,Y 467.573,Z 262.152,A -85,B 0,C 180,E1 -7796.011,E2 -7796.011} C_VEL
LIN {X 0,Y 467.669,Z 270.881,A -85,B 0,C 180,E1 -7798.021,E2 -7798.021} C_VEL
LIN {X 0,Y 467.625,Z 277.826,A -85,B 0,C 180,E1 -7799.612,E2 -7799.612} C_VEL
LIN {X 0,Y 469.768,Z 290.422,A -85,B 0,C 180,E1 -7799.892,E2 -7799.892} C_VEL
LIN {X 0,Y 469.275,Z 354.625,A -85,B 0,C 180,E1 -7800.905,E2 -7800.905} C_VEL
LIN {X 0,Y 469.107,Z 365.382,A -85,B 0,C 180,E1 -7801.215,E2 -7801.215} C_VEL
LIN {X 0,Y 468.88,Z 377.406,A -85,B 0,C 180,E1 -7801.766,E2 -7801.766} C_VEL
LIN {X 0,Y 468.597,Z 385.921,A -85,B 0,C 180,E1 -7802.294,E2 -7802.294} C_VEL
LIN {X 0,Y 468.523,Z 388.76,A -85,B 0,C 180,E1 -7802.501,E2 -7802.501} C_VEL
LIN {X 0,Y 467.67,Z 393.783,A -85,B 0,C 180,E1 -7802.872,E2 -7802.872} C_VEL
LIN {X 0,Y 464.503,Z 401.605,A -85,B 0,C 180,E1 -7803.521,E2 -7803.521} C_VEL
LIN {X 0,Y 461.37,Z 408.735,A -85,B 0,C 180,E1 -7804.278,E2 -7804.278} C_VEL
LIN {X 0,Y 460.575,Z 412.664,A -85,B 0,C 180,E1 -7804.815,E2 -7804.815} C_VEL
LIN {X 0,Y 460.296,Z 419.101,A -85,B 0,C 180,E1 -7805.862,E2 -7805.862} C_VEL
LIN {X 0,Y 460.082,Z 423.979,A -85,B 0,C 180,E1 -7806.837,E2 -7806.837} C_VEL
LIN {X 0,Y 459.955,Z 426.995,A -85,B 0,C 180,E1 -7807.543,E2 -7807.543} C_VEL
LIN {X 0,Y 459.795,Z 431.137,A -85,B 0,C 180,E1 -7808.797,E2 -7808.797} C_VEL
LIN {X 0,Y 459.753,Z 432.739,A -85,B 0,C 180,E1 -7809.416,E2 -7809.416} C_VEL
LIN {X 0,Y 459.613,Z 434.618,A -85,B 0,C 180,E1 -7810.342,E2 -7810.342} C_VEL
LIN {X 0,Y 459.547,Z 436.134,A -85,B 0,C 180,E1 -7811.46,E2 -7811.46} C_VEL
LIN {X 0,Y 459.543,Z 436.692,A -85,B 0,C 180,E1 -7812.19,E2 -7812.19} C_VEL
LIN {X 0,Y 459.536,Z 436.939,A -85,B 0,C 180,E1 -7813.107,E2 -7813.107} C_VEL
LIN {X 0,Y 459.593,Z 436.227,A -85,B 0,C 180,E1 -7814.429,E2 -7814.429} C_VEL
LIN {X 0,Y 459.604,Z 434.238,A -85,B 0,C 180,E1 -7815.838,E2 -7815.838} C_VEL
LIN {X 0,Y 459.76,Z 431.075,A -85,B 0,C 180,E1 -7817.194,E2 -7817.194} C_VEL
LIN {X 0,Y 459.902,Z 426.527,A -85,B 0,C 180,E1 -7818.542,E2 -7818.542} C_VEL
LIN {X 0,Y 460.128,Z 421.446,A -85,B 0,C 180,E1 -7819.661,E2 -7819.661} C_VEL
LIN {X 0,Y 460.283,Z 416.506,A -85,B 0,C 180,E1 -7820.553,E2 -7820.553} C_VEL
LIN {X 0,Y 460.514,Z 410.529,A -85,B 0,C 180,E1 -7821.443,E2 -7821.443} C_VEL
LIN {X 0,Y 460.886,Z 403.086,A -85,B 0,C 180,E1 -7822.347,E2 -7822.347} C_VEL
LIN {X 0,Y 461.14,Z 395.458,A -85,B 0,C 180,E1 -7823.107,E2 -7823.107} C_VEL
LIN {X 0,Y 461.448,Z 387.262,A -85,B 0,C 180,E1 -7823.77,E2 -7823.77} C_VEL
LIN {X 0,Y 461.7,Z 378.74,A -85,B 0,C 180,E1 -7824.322,E2 -7824.322} C_VEL
LIN {X 0,Y 461.924,Z 368.776,A -85,B 0,C 180,E1 -7824.817,E2 -7824.817} C_VEL
LIN {X 0,Y 462.116,Z 356.208,A -85,B 0,C 180,E1 -7825.229,E2 -7825.229} C_VEL
LIN {X 0,Y 462.262,Z 335.555,A -85,B 0,C 180,E1 -7825.586,E2 -7825.586} C_VEL
LIN {X 0,Y 462.444,Z 289.102,A -85,B 0,C 180,E1 -7826.311,E2 -7826.311} C_VEL
LIN {X 0,Y 460.432,Z 278.127,A -85,B 0,C 180,E1 -7826.555,E2 -7826.555} C_VEL
LIN {X 0,Y 460.707,Z 265.557,A -85,B 0,C 180,E1 -7829.563,E2 -7829.563} C_VEL
LIN {X 0,Y 460.634,Z 262.919,A -85,B 0,C 180,E1 -7830.219,E2 -7830.219} C_VEL
LIN {X 0,Y 460.787,Z 262.897,A -85,B 0,C 180,E1 -7832.623,E2 -7832.623} C_VEL
LIN {X 0,Y 460.666,Z 262.911,A -85,B 0,C 180,E1 -7836.131,E2 -7836.131} C_VEL
LIN {X 0,Y 460.591,Z 262.922,A -85,B 0,C 180,E1 -7838.777,E2 -7838.777} C_VEL
LIN {X 0,Y 460.577,Z 262.922,A -85,B 0,C 180,E1 -7842.446,E2 -7842.446} C_VEL
LIN {X 0,Y 460.564,Z 262.924,A -85,B 0,C 180,E1 -7845.999,E2 -7845.999} C_VEL
LIN {X 0,Y 460.535,Z 262.929,A -85,B 0,C 180,E1 -7848.903,E2 -7848.903} C_VEL
LIN {X 0,Y 460.481,Z 262.94,A -85,B 0,C 180,E1 -7851.488,E2 -7851.488} C_VEL
LIN {X 0,Y 460.486,Z 262.932,A -85,B 0,C 180,E1 -7854.336,E2 -7854.336} C_VEL
LIN {X 0,Y 460.501,Z 262.936,A -85,B 0,C 180,E1 -7857.249,E2 -7857.249} C_VEL
LIN {X 0,Y 460.475,Z 262.934,A -85,B 0,C 180,E1 -7860.243,E2 -7860.243} C_VEL
LIN {X 0,Y 460.497,Z 262.937,A -85,B 0,C 180,E1 -7863.328,E2 -7863.328} C_VEL
LIN {X 0,Y 460.444,Z 262.938,A -85,B 0,C 180,E1 -7866.533,E2 -7866.533} C_VEL
LIN {X 0,Y 460.487,Z 262.937,A -85,B 0,C 180,E1 -7869.867,E2 -7869.867} C_VEL
LIN {X 0,Y 460.467,Z 262.936,A -85,B 0,C 180,E1 -7872.901,E2 -7872.901} C_VEL
LIN {X 0,Y 460.484,Z 262.939,A -85,B 0,C 180,E1 -7875.834,E2 -7875.834} C_VEL
LIN {X 0,Y 460.51,Z 262.931,A -85,B 0,C 180,E1 -7878.992,E2 -7878.992} C_VEL
LIN {X 0,Y 460.499,Z 262.934,A -85,B 0,C 180,E1 -7881.27,E2 -7881.27} C_VEL
LIN {X 0,Y 460.491,Z 262.933,A -85,B 0,C 180,E1 -7884.558,E2 -7884.558} C_VEL
LIN {X 0,Y 460.515,Z 262.936,A -85,B 0,C 180,E1 -7887.719,E2 -7887.719} C_VEL
LIN {X 0,Y 460.513,Z 262.93,A -85,B 0,C 180,E1 -7890.772,E2 -7890.772} C_VEL
LIN {X 0,Y 460.516,Z 262.936,A -85,B 0,C 180,E1 -7893.736,E2 -7893.736} C_VEL
LIN {X 0,Y 460.534,Z 262.928,A -85,B 0,C 180,E1 -7896.627,E2 -7896.627} C_VEL
LIN {X 0,Y 460.542,Z 262.929,A -85,B 0,C 180,E1 -7899.456,E2 -7899.456} C_VEL
LIN {X 0,Y 460.539,Z 262.931,A -85,B 0,C 180,E1 -7902.233,E2 -7902.233} C_VEL
LIN {X 0,Y 460.584,Z 263.128,A -85,B 0,C 180,E1 -7903.036,E2 -7903.036} C_VEL
LIN {X 0,Y 460.51,Z 272.923,A -85,B 0,C 180,E1 -7905.419,E2 -7905.419} C_VEL
LIN {X 0,Y 460.438,Z 277.915,A -85,B 0,C 180,E1 -7906.627,E2 -7906.627} C_VEL
LIN {X 0,Y 462.417,Z 290.371,A -85,B 0,C 180,E1 -7906.904,E2 -7906.904} C_VEL
LIN {X 0,Y 461.813,Z 355.228,A -85,B 0,C 180,E1 -7908.064,E2 -7908.064} C_VEL
LIN {X 0,Y 461.658,Z 364.938,A -85,B 0,C 180,E1 -7908.366,E2 -7908.366} C_VEL
LIN {X 0,Y 461.425,Z 374.837,A -85,B 0,C 180,E1 -7908.806,E2 -7908.806} C_VEL
LIN {X 0,Y 461.232,Z 385.866,A -85,B 0,C 180,E1 -7909.467,E2 -7909.467} C_VEL
LIN {X 0,Y 460.928,Z 395.416,A -85,B 0,C 180,E1 -7910.237,E2 -7910.237} C_VEL
LIN {X 0,Y 460.667,Z 403.135,A -85,B 0,C 180,E1 -7911.007,E2 -7911.007} C_VEL
LIN {X 0,Y 460.393,Z 410.386,A -85,B 0,C 180,E1 -7911.886,E2 -7911.886} C_VEL
LIN {X 0,Y 460.226,Z 418.002,A -85,B 0,C 180,E1 -7913.028,E2 -7913.028} C_VEL
LIN {X 0,Y 459.945,Z 424.47,A -85,B 0,C 180,E1 -7914.303,E2 -7914.303} C_VEL
LIN {X 0,Y 459.839,Z 429.562,A -85,B 0,C 180,E1 -7915.62,E2 -7915.62} C_VEL
LIN {X 0,Y 459.793,Z 432.114,A -85,B 0,C 180,E1 -7916.498,E2 -7916.498} C_VEL
LIN {X 0,Y 459.671,Z 434.089,A -85,B 0,C 180,E1 -7917.374,E2 -7917.374} C_VEL
LIN {X 0,Y 459.607,Z 435.527,A -85,B 0,C 180,E1 -7918.25,E2 -7918.25} C_VEL
LIN {X 0,Y 459.56,Z 436.454,A -85,B 0,C 180,E1 -7919.127,E2 -7919.127} C_VEL
LIN {X 0,Y 459.542,Z 436.813,A -85,B 0,C 180,E1 -7920.003,E2 -7920.003} C_VEL
LIN {X 0,Y 459.561,Z 436.602,A -85,B 0,C 180,E1 -7920.879,E2 -7920.879} C_VEL
LIN {X 0,Y 459.64,Z 435.888,A -85,B 0,C 180,E1 -7921.755,E2 -7921.755} C_VEL
LIN {X 0,Y 459.708,Z 434.667,A -85,B 0,C 180,E1 -7922.631,E2 -7922.631} C_VEL
LIN {X 0,Y 459.844,Z 431.784,A -85,B 0,C 180,E1 -7923.946,E2 -7923.946} C_VEL
LIN {X 0,Y 459.939,Z 429.109,A -85,B 0,C 180,E1 -7924.824,E2 -7924.824} C_VEL
LIN {X 0,Y 459.951,Z 425.794,A -85,B 0,C 180,E1 -7925.703,E2 -7925.703} C_VEL
LIN {X 0,Y 460.254,Z 421.096,A -85,B 0,C 180,E1 -7926.704,E2 -7926.704} C_VEL
LIN {X 0,Y 460.355,Z 415.504,A -85,B 0,C 180,E1 -7927.679,E2 -7927.679} C_VEL
LIN {X 0,Y 460.654,Z 407.697,A -85,B 0,C 180,E1 -7928.778,E2 -7928.778} C_VEL
LIN {X 0,Y 461.02,Z 398.579,A -85,B 0,C 180,E1 -7929.767,E2 -7929.767} C_VEL
LIN {X 0,Y 461.336,Z 391.075,A -85,B 0,C 180,E1 -7930.425,E2 -7930.425} C_VEL
LIN {X 0,Y 461.544,Z 383.482,A -85,B 0,C 180,E1 -7930.975,E2 -7930.975} C_VEL
LIN {X 0,Y 461.769,Z 373.889,A -85,B 0,C 180,E1 -7931.525,E2 -7931.525} C_VEL
LIN {X 0,Y 461.982,Z 362.851,A -85,B 0,C 180,E1 -7931.993,E2 -7931.993} C_VEL
LIN {X 0,Y 462.205,Z 350.228,A -85,B 0,C 180,E1 -7932.314,E2 -7932.314} C_VEL
LIN {X 0,Y 462.776,Z 289.704,A -85,B 0,C 180,E1 -7933.429,E2 -7933.429} C_VEL
LIN {X 0,Y 460.693,Z 279.074,A -85,B 0,C 180,E1 -7933.729,E2 -7933.729} C_VEL
LIN {X 0,Y 460.844,Z 266.879,A -85,B 0,C 180,E1 -7936.595,E2 -7936.595} C_VEL
LIN {X 0,Y 460.625,Z 262.928,A -85,B 0,C 180,E1 -7937.54,E2 -7937.54} C_VEL
LIN {X 0,Y 460.559,Z 262.931,A -85,B 0,C 180,E1 -7940.549,E2 -7940.549} C_VEL
LIN {X 0,Y 460.535,Z 262.93,A -85,B 0,C 180,E1 -7943.704,E2 -7943.704} C_VEL
LIN {X 0,Y 460.528,Z 262.935,A -85,B 0,C 180,E1 -7946.27,E2 -7946.27} C_VEL
LIN {X 0,Y 460.534,Z 262.929,A -85,B 0,C 180,E1 -7949.233,E2 -7949.233} C_VEL
LIN {X 0,Y 460.538,Z 262.934,A -85,B 0,C 180,E1 -7952.286,E2 -7952.286} C_VEL
LIN {X 0,Y 460.515,Z 262.931,A -85,B 0,C 180,E1 -7955.447,E2 -7955.447} C_VEL
LIN {X 0,Y 460.512,Z 262.934,A -85,B 0,C 180,E1 -7958.892,E2 -7958.892} C_VEL
LIN {X 0,Y 460.521,Z 262.93,A -85,B 0,C 180,E1 -7961.601,E2 -7961.601} C_VEL
LIN {X 0,Y 460.52,Z 262.934,A -85,B 0,C 180,E1 -7964.59,E2 -7964.59} C_VEL
LIN {X 0,Y 460.512,Z 262.93,A -85,B 0,C 180,E1 -7967.817,E2 -7967.817} C_VEL
LIN {X 0,Y 460.526,Z 262.931,A -85,B 0,C 180,E1 -7970.137,E2 -7970.137} C_VEL
LIN {X 0,Y 460.48,Z 262.932,A -85,B 0,C 180,E1 -7973.471,E2 -7973.471} C_VEL
LIN {X 0,Y 460.524,Z 262.933,A -85,B 0,C 180,E1 -7976.674,E2 -7976.674} C_VEL
LIN {X 0,Y 460.516,Z 262.931,A -85,B 0,C 180,E1 -7979.76,E2 -7979.76} C_VEL
LIN {X 0,Y 460.575,Z 262.927,A -85,B 0,C 180,E1 -7982.756,E2 -7982.756} C_VEL
LIN {X 0,Y 460.616,Z 263.103,A -85,B 0,C 180,E1 -7985.612,E2 -7985.612} C_VEL
LIN {X 0,Y 461.883,Z 270.61,A -85,B 0,C 180,E1 -7987.169,E2 -7987.169} C_VEL
LIN {X 0,Y 461.537,Z 281.24,A -85,B 0,C 180,E1 -7989.265,E2 -7989.265} C_VEL
LIN {X 0,Y 460.992,Z 296.533,A -85,B 0,C 180,E1 -7992.247,E2 -7992.247} C_VEL
LIN {X 0,Y 460.462,Z 314.087,A -85,B 0,C 180,E1 -7995.639,E2 -7995.639} C_VEL
LIN {X 0,Y 460.375,Z 318.345,A -85,B 0,C 180,E1 -7996.459,E2 -7996.459} C_VEL
LIN {X 0,Y 462.412,Z 337.031,A -85,B 0,C 180,E1 -7996.822,E2 -7996.822} C_VEL
LIN {X 0,Y 462.066,Z 395.981,A -85,B 0,C 180,E1 -7997.761,E2 -7997.761} C_VEL
LIN {X 0,Y 461.782,Z 405.776,A -85,B 0,C 180,E1 -7998.032,E2 -7998.032} C_VEL
LIN {X 0,Y 461.448,Z 417.454,A -85,B 0,C 180,E1 -7998.524,E2 -7998.524} C_VEL
LIN {X 0,Y 461.143,Z 427.411,A -85,B 0,C 180,E1 -7999.129,E2 -7999.129} C_VEL
LIN {X 0,Y 460.808,Z 435.919,A -85,B 0,C 180,E1 -7999.787,E2 -7999.787} C_VEL
LIN {X 0,Y 460.521,Z 443.947,A -85,B 0,C 180,E1 -8000.557,E2 -8000.557} C_VEL
LIN {X 0,Y 460.291,Z 449.714,A -85,B 0,C 180,E1 -8001.217,E2 -8001.217} C_VEL
LIN {X 0,Y 460.037,Z 456.152,A -85,B 0,C 180,E1 -8002.097,E2 -8002.097} C_VEL
LIN {X 0,Y 459.943,Z 461.509,A -85,B 0,C 180,E1 -8002.978,E2 -8002.978} C_VEL
LIN {X 0,Y 459.728,Z 465.969,A -85,B 0,C 180,E1 -8003.857,E2 -8003.857} C_VEL
LIN {X 0,Y 459.71,Z 469.69,A -85,B 0,C 180,E1 -8004.737,E2 -8004.737} C_VEL
LIN {X 0,Y 459.587,Z 472.721,A -85,B 0,C 180,E1 -8005.615,E2 -8005.615} C_VEL
LIN {X 0,Y 459.654,Z 475.079,A -85,B 0,C 180,E1 -8006.493,E2 -8006.493} C_VEL
LIN {X 0,Y 459.61,Z 476.868,A -85,B 0,C 180,E1 -8007.371,E2 -8007.371} C_VEL
LIN {X 0,Y 459.572,Z 478.153,A -85,B 0,C 180,E1 -8008.247,E2 -8008.247} C_VEL
LIN {X 0,Y 459.556,Z 478.961,A -85,B 0,C 180,E1 -8009.124,E2 -8009.124} C_VEL
LIN {X 0,Y 459.537,Z 479.262,A -85,B 0,C 180,E1 -8010,E2 -8010} C_VEL
LIN {X 0,Y 459.556,Z 478.974,A -85,B 0,C 180,E1 -8010.876,E2 -8010.876} C_VEL
LIN {X 0,Y 459.572,Z 478.208,A -85,B 0,C 180,E1 -8011.752,E2 -8011.752} C_VEL
LIN {X 0,Y 459.61,Z 476.967,A -85,B 0,C 180,E1 -8012.629,E2 -8012.629} C_VEL
LIN {X 0,Y 459.652,Z 475.228,A -85,B 0,C 180,E1 -8013.506,E2 -8013.506} C_VEL
LIN {X 0,Y 459.649,Z 471.422,A -85,B 0,C 180,E1 -8014.824,E2 -8014.824} C_VEL
LIN {X 0,Y 459.73,Z 466.237,A -85,B 0,C 180,E1 -8016.143,E2 -8016.143} C_VEL
LIN {X 0,Y 459.962,Z 460.677,A -85,B 0,C 180,E1 -8017.242,E2 -8017.242} C_VEL
LIN {X 0,Y 460.165,Z 453.714,A -85,B 0,C 180,E1 -8018.342,E2 -8018.342} C_VEL
LIN {X 0,Y 460.508,Z 445.741,A -85,B 0,C 180,E1 -8019.332,E2 -8019.332} C_VEL
LIN {X 0,Y 460.839,Z 438.144,A -85,B 0,C 180,E1 -8020.101,E2 -8020.101} C_VEL
LIN {X 0,Y 461.138,Z 430.197,A -85,B 0,C 180,E1 -8020.76,E2 -8020.76} C_VEL
LIN {X 0,Y 461.435,Z 422.015,A -85,B 0,C 180,E1 -8021.309,E2 -8021.309} C_VEL
LIN {X 0,Y 461.709,Z 413.753,A -85,B 0,C 180,E1 -8021.747,E2 -8021.747} C_VEL
LIN {X 0,Y 461.976,Z 404.87,A -85,B 0,C 180,E1 -8022.102,E2 -8022.102} C_VEL
LIN {X 0,Y 462.272,Z 395.952,A -85,B 0,C 180,E1 -8022.346,E2 -8022.346} C_VEL
LIN {X 0,Y 462.514,Z 335.137,A -85,B 0,C 180,E1 -8023.326,E2 -8023.326} C_VEL
LIN {X 0,Y 460.408,Z 318.01,A -85,B 0,C 180,E1 -8023.686,E2 -8023.686} C_VEL
LIN {X 0,Y 460.821,Z 302.936,A -85,B 0,C 180,E1 -8026.593,E2 -8026.593} C_VEL
LIN {X 0,Y 461.492,Z 286.455,A -85,B 0,C 180,E1 -8029.806,E2 -8029.806} C_VEL
LIN {X 0,Y 461.989,Z 272.387,A -85,B 0,C 180,E1 -8032.589,E2 -8032.589} C_VEL
LIN {X 0,Y 461.171,Z 266.19,A -85,B 0,C 180,E1 -8033.882,E2 -8033.882} C_VEL
LIN {X 0,Y 460.558,Z 262.932,A -85,B 0,C 180,E1 -8034.601,E2 -8034.601} C_VEL
LIN {X 0,Y 460.586,Z 262.924,A -85,B 0,C 180,E1 -8037.745,E2 -8037.745} C_VEL
LIN {X 0,Y 460.526,Z 262.935,A -85,B 0,C 180,E1 -8041.282,E2 -8041.282} C_VEL
LIN {X 0,Y 460.529,Z 262.93,A -85,B 0,C 180,E1 -8044.503,E2 -8044.503} C_VEL
LIN {X 0,Y 460.507,Z 262.937,A -85,B 0,C 180,E1 -8047.622,E2 -8047.622} C_VEL
LIN {X 0,Y 460.536,Z 262.93,A -85,B 0,C 180,E1 -8051.011,E2 -8051.011} C_VEL
LIN {X 0,Y 460.519,Z 262.927,A -85,B 0,C 180,E1 -8054.588,E2 -8054.588} C_VEL
LIN {X 0,Y 460.511,Z 262.934,A -85,B 0,C 180,E1 -8057.815,E2 -8057.815} C_VEL
LIN {X 0,Y 460.524,Z 262.928,A -85,B 0,C 180,E1 -8060.135,E2 -8060.135} C_VEL
LIN {X 0,Y 460.482,Z 262.94,A -85,B 0,C 180,E1 -8063.469,E2 -8063.469} C_VEL
LIN {X 0,Y 460.526,Z 262.928,A -85,B 0,C 180,E1 -8066.673,E2 -8066.673} C_VEL
LIN {X 0,Y 460.513,Z 262.934,A -85,B 0,C 180,E1 -8069.758,E2 -8069.758} C_VEL
LIN {X 0,Y 460.541,Z 262.924,A -85,B 0,C 180,E1 -8072.752,E2 -8072.752} C_VEL
LIN {X 0,Y 460.535,Z 262.933,A -85,B 0,C 180,E1 -8075.665,E2 -8075.665} C_VEL
LIN {X 0,Y 460.527,Z 262.923,A -85,B 0,C 180,E1 -8078.576,E2 -8078.576} C_VEL
LIN {X 0,Y 460.59,Z 262.921,A -85,B 0,C 180,E1 -8081.309,E2 -8081.309} C_VEL
LIN {X 0,Y 460.609,Z 262.919,A -85,B 0,C 180,E1 -8084.057,E2 -8084.057} C_VEL
LIN {X 0,Y 460.614,Z 262.92,A -85,B 0,C 180,E1 -8087.664,E2 -8087.664} C_VEL
LIN {X 0,Y 460.63,Z 262.913,A -85,B 0,C 180,E1 -8091.221,E2 -8091.221} C_VEL
LIN {X 0,Y 460.705,Z 262.907,A -85,B 0,C 180,E1 -8093.867,E2 -8093.867} C_VEL
LIN {X 0,Y 460.79,Z 262.894,A -85,B 0,C 180,E1 -8097.375,E2 -8097.375} C_VEL
LIN {X 0,Y 460.85,Z 262.887,A -85,B 0,C 180,E1 -8099.997,E2 -8099.997} C_VEL
LIN {X 0,Y 460.791,Z 262.895,A -85,B 0,C 180,E1 -8102.62,E2 -8102.62} C_VEL
LIN {X 0,Y 460.68,Z 262.91,A -85,B 0,C 180,E1 -8106.127,E2 -8106.127} C_VEL
LIN {X 0,Y 460.616,Z 262.917,A -85,B 0,C 180,E1 -8108.773,E2 -8108.773} C_VEL
LIN {X 0,Y 460.608,Z 262.924,A -85,B 0,C 180,E1 -8112.442,E2 -8112.442} C_VEL
LIN {X 0,Y 460.593,Z 262.92,A -85,B 0,C 180,E1 -8115.994,E2 -8115.994} C_VEL
LIN {X 0,Y 460.559,Z 262.923,A -85,B 0,C 180,E1 -8119.612,E2 -8119.612} C_VEL
LIN {X 0,Y 460.5,Z 262.939,A -85,B 0,C 180,E1 -8122.425,E2 -8122.425} C_VEL
LIN {X 0,Y 460.555,Z 262.924,A -85,B 0,C 180,E1 -8125.799,E2 -8125.799} C_VEL
LIN {X 0,Y 460.538,Z 262.931,A -85,B 0,C 180,E1 -8128.23,E2 -8128.23} C_VEL
LIN {X 0,Y 460.505,Z 262.93,A -85,B 0,C 180,E1 -8131.28,E2 -8131.28} C_VEL
LIN {X 0,Y 460.515,Z 262.933,A -85,B 0,C 180,E1 -8134.503,E2 -8134.503} C_VEL
LIN {X 0,Y 460.481,Z 262.934,A -85,B 0,C 180,E1 -8137.62,E2 -8137.62} C_VEL
LIN {X 0,Y 460.521,Z 262.931,A -85,B 0,C 180,E1 -8140.266,E2 -8140.266} C_VEL
LIN {X 0,Y 460.501,Z 262.931,A -85,B 0,C 180,E1 -8143.369,E2 -8143.369} C_VEL
LIN {X 0,Y 460.5,Z 262.937,A -85,B 0,C 180,E1 -8146.625,E2 -8146.625} C_VEL
LIN {X 0,Y 460.533,Z 262.929,A -85,B 0,C 180,E1 -8149.725,E2 -8149.725} C_VEL
LIN {X 0,Y 460.501,Z 262.939,A -85,B 0,C 180,E1 -8152.516,E2 -8152.516} C_VEL
LIN {X 0,Y 460.562,Z 263.083,A -85,B 0,C 180,E1 -8155.89,E2 -8155.89} C_VEL
LIN {X 0,Y 460.72,Z 270.991,A -85,B 0,C 180,E1 -8157.731,E2 -8157.731} C_VEL
LIN {X 0,Y 460.627,Z 278.21,A -85,B 0,C 180,E1 -8159.396,E2 -8159.396} C_VEL
LIN {X 0,Y 462.906,Z 291.309,A -85,B 0,C 180,E1 -8159.681,E2 -8159.681} C_VEL
LIN {X 0,Y 462.393,Z 354.35,A -85,B 0,C 180,E1 -8160.688,E2 -8160.688} C_VEL
LIN {X 0,Y 462.254,Z 363.72,A -85,B 0,C 180,E1 -8160.95,E2 -8160.95} C_VEL
LIN {X 0,Y 462.037,Z 373.879,A -85,B 0,C 180,E1 -8161.371,E2 -8161.371} C_VEL
LIN {X 0,Y 461.783,Z 384.191,A -85,B 0,C 180,E1 -8161.962,E2 -8161.962} C_VEL
LIN {X 0,Y 461.439,Z 393.674,A -85,B 0,C 180,E1 -8162.691,E2 -8162.691} C_VEL
LIN {X 0,Y 461.077,Z 401.15,A -85,B 0,C 180,E1 -8163.401,E2 -8163.401} C_VEL
LIN {X 0,Y 460.814,Z 407.492,A -85,B 0,C 180,E1 -8164.124,E2 -8164.124} C_VEL
LIN {X 0,Y 460.575,Z 412.664,A -85,B 0,C 180,E1 -8164.815,E2 -8164.815} C_VEL
LIN {X 0,Y 459.793,Z 416.466,A -85,B 0,C 180,E1 -8165.384,E2 -8165.384} C_VEL
LIN {X 0,Y 456.683,Z 422.076,A -85,B 0,C 180,E1 -8166.332,E2 -8166.332} C_VEL
LIN {X 0,Y 453.583,Z 426.911,A -85,B 0,C 180,E1 -8167.35,E2 -8167.35} C_VEL
LIN {X 0,Y 452.812,Z 429.315,A -85,B 0,C 180,E1 -8168.019,E2 -8168.019} C_VEL
LIN {X 0,Y 452.687,Z 432.409,A -85,B 0,C 180,E1 -8169.079,E2 -8169.079} C_VEL
LIN {X 0,Y 452.576,Z 434.488,A -85,B 0,C 180,E1 -8170.024,E2 -8170.024} C_VEL
LIN {X 0,Y 452.48,Z 436.372,A -85,B 0,C 180,E1 -8171.33,E2 -8171.33} C_VEL
LIN {X 0,Y 452.451,Z 436.925,A -85,B 0,C 180,E1 -8171.901,E2 -8171.901} C_VEL
LIN {X 0,Y 452.437,Z 437.257,A -85,B 0,C 180,E1 -8172.834,E2 -8172.834} C_VEL
LIN {X 0,Y 452.495,Z 436.652,A -85,B 0,C 180,E1 -8174.339,E2 -8174.339} C_VEL
LIN {X 0,Y 452.516,Z 435.015,A -85,B 0,C 180,E1 -8175.612,E2 -8175.612} C_VEL
LIN {X 0,Y 452.64,Z 432.042,A -85,B 0,C 180,E1 -8176.989,E2 -8176.989} C_VEL
LIN {X 0,Y 452.767,Z 429.298,A -85,B 0,C 180,E1 -8177.91,E2 -8177.91} C_VEL
LIN {X 0,Y 452.963,Z 424.014,A -85,B 0,C 180,E1 -8179.27,E2 -8179.27} C_VEL
LIN {X 0,Y 453.23,Z 416.951,A -85,B 0,C 180,E1 -8180.63,E2 -8180.63} C_VEL
LIN {X 0,Y 453.49,Z 410.991,A -85,B 0,C 180,E1 -8181.534,E2 -8181.534} C_VEL
LIN {X 0,Y 453.796,Z 404.549,A -85,B 0,C 180,E1 -8182.346,E2 -8182.346} C_VEL
LIN {X 0,Y 454.05,Z 397.236,A -85,B 0,C 180,E1 -8183.11,E2 -8183.11} C_VEL
LIN {X 0,Y 454.416,Z 389.332,A -85,B 0,C 180,E1 -8183.785,E2 -8183.785} C_VEL
LIN {X 0,Y 454.658,Z 381.252,A -85,B 0,C 180,E1 -8184.345,E2 -8184.345} C_VEL
LIN {X 0,Y 454.887,Z 371.923,A -85,B 0,C 180,E1 -8184.848,E2 -8184.848} C_VEL
LIN {X 0,Y 455.083,Z 362.798,A -85,B 0,C 180,E1 -8185.211,E2 -8185.211} C_VEL
LIN {X 0,Y 455.218,Z 353.466,A -85,B 0,C 180,E1 -8185.462,E2 -8185.462} C_VEL
LIN {X 0,Y 455.582,Z 290.345,A -85,B 0,C 180,E1 -8186.476,E2 -8186.476} C_VEL
LIN {X 0,Y 453.41,Z 278.377,A -85,B 0,C 180,E1 -8186.751,E2 -8186.751} C_VEL
LIN {X 0,Y 453.687,Z 266.764,A -85,B 0,C 180,E1 -8189.556,E2 -8189.556} C_VEL
LIN {X 0,Y 453.632,Z 263.792,A -85,B 0,C 180,E1 -8190.333,E2 -8190.333} C_VEL
LIN {X 0,Y 453.727,Z 263.777,A -85,B 0,C 180,E1 -8192.664,E2 -8192.664} C_VEL
LIN {X 0,Y 453.634,Z 263.787,A -85,B 0,C 180,E1 -8196.226,E2 -8196.226} C_VEL
LIN {X 0,Y 453.554,Z 263.8,A -85,B 0,C 180,E1 -8198.914,E2 -8198.914} C_VEL
LIN {X 0,Y 453.527,Z 263.8,A -85,B 0,C 180,E1 -8202.53,E2 -8202.53} C_VEL
LIN {X 0,Y 453.509,Z 263.802,A -85,B 0,C 180,E1 -8206.197,E2 -8206.197} C_VEL
LIN {X 0,Y 453.484,Z 263.808,A -85,B 0,C 180,E1 -8209.042,E2 -8209.042} C_VEL
LIN {X 0,Y 453.442,Z 263.813,A -85,B 0,C 180,E1 -8211.838,E2 -8211.838} C_VEL
LIN {X 0,Y 453.459,Z 263.808,A -85,B 0,C 180,E1 -8214.738,E2 -8214.738} C_VEL
LIN {X 0,Y 453.458,Z 263.81,A -85,B 0,C 180,E1 -8217.952,E2 -8217.952} C_VEL
LIN {X 0,Y 453.444,Z 263.81,A -85,B 0,C 180,E1 -8220.762,E2 -8220.762} C_VEL
LIN {X 0,Y 453.446,Z 263.813,A -85,B 0,C 180,E1 -8223.916,E2 -8223.916} C_VEL
LIN {X 0,Y 453.421,Z 263.816,A -85,B 0,C 180,E1 -8227.193,E2 -8227.193} C_VEL
LIN {X 0,Y 453.445,Z 263.81,A -85,B 0,C 180,E1 -8230.615,E2 -8230.615} C_VEL
LIN {X 0,Y 453.436,Z 263.812,A -85,B 0,C 180,E1 -8234.225,E2 -8234.225} C_VEL
LIN {X 0,Y 453.439,Z 263.812,A -85,B 0,C 180,E1 -8237.008,E2 -8237.008} C_VEL
LIN {X 0,Y 453.474,Z 263.811,A -85,B 0,C 180,E1 -8239.412,E2 -8239.412} C_VEL
LIN {X 0,Y 453.433,Z 263.812,A -85,B 0,C 180,E1 -8242.814,E2 -8242.814} C_VEL
LIN {X 0,Y 453.452,Z 263.813,A -85,B 0,C 180,E1 -8246.09,E2 -8246.09} C_VEL
LIN {X 0,Y 453.461,Z 263.81,A -85,B 0,C 180,E1 -8249.244,E2 -8249.244} C_VEL
LIN {X 0,Y 453.495,Z 263.806,A -85,B 0,C 180,E1 -8252.299,E2 -8252.299} C_VEL
LIN {X 0,Y 453.484,Z 263.807,A -85,B 0,C 180,E1 -8255.268,E2 -8255.268} C_VEL
LIN {X 0,Y 453.472,Z 263.809,A -85,B 0,C 180,E1 -8258.419,E2 -8258.419} C_VEL
LIN {X 0,Y 453.516,Z 263.802,A -85,B 0,C 180,E1 -8261.012,E2 -8261.012} C_VEL
LIN {X 0,Y 453.552,Z 263.967,A -85,B 0,C 180,E1 -8262.997,E2 -8262.997} C_VEL
LIN {X 0,Y 453.455,Z 274.835,A -85,B 0,C 180,E1 -8265.645,E2 -8265.645} C_VEL
LIN {X 0,Y 453.432,Z 278.207,A -85,B 0,C 180,E1 -8266.445,E2 -8266.445} C_VEL
LIN {X 0,Y 455.448,Z 290.996,A -85,B 0,C 180,E1 -8266.738,E2 -8266.738} C_VEL
LIN {X 0,Y 454.83,Z 355.017,A -85,B 0,C 180,E1 -8267.906,E2 -8267.906} C_VEL
LIN {X 0,Y 454.644,Z 365.567,A -85,B 0,C 180,E1 -8268.241,E2 -8268.241} C_VEL
LIN {X 0,Y 454.419,Z 375.379,A -85,B 0,C 180,E1 -8268.687,E2 -8268.687} C_VEL
LIN {X 0,Y 454.239,Z 385.537,A -85,B 0,C 180,E1 -8269.303,E2 -8269.303} C_VEL
LIN {X 0,Y 453.921,Z 395.255,A -85,B 0,C 180,E1 -8270.085,E2 -8270.085} C_VEL
LIN {X 0,Y 453.659,Z 403.053,A -85,B 0,C 180,E1 -8270.866,E2 -8270.866} C_VEL
LIN {X 0,Y 453.353,Z 410.373,A -85,B 0,C 180,E1 -8271.759,E2 -8271.759} C_VEL
LIN {X 0,Y 453.164,Z 417.814,A -85,B 0,C 180,E1 -8272.876,E2 -8272.876} C_VEL
LIN {X 0,Y 452.941,Z 423.654,A -85,B 0,C 180,E1 -8273.991,E2 -8273.991} C_VEL
LIN {X 0,Y 452.774,Z 428.222,A -85,B 0,C 180,E1 -8275.106,E2 -8275.106} C_VEL
LIN {X 0,Y 452.731,Z 432.335,A -85,B 0,C 180,E1 -8276.443,E2 -8276.443} C_VEL
LIN {X 0,Y 452.596,Z 434.343,A -85,B 0,C 180,E1 -8277.333,E2 -8277.333} C_VEL
LIN {X 0,Y 452.519,Z 435.811,A -85,B 0,C 180,E1 -8278.223,E2 -8278.223} C_VEL
LIN {X 0,Y 452.495,Z 436.758,A -85,B 0,C 180,E1 -8279.113,E2 -8279.113} C_VEL
LIN {X 0,Y 452.475,Z 437.127,A -85,B 0,C 180,E1 -8280.003,E2 -8280.003} C_VEL
LIN {X 0,Y 452.497,Z 436.936,A -85,B 0,C 180,E1 -8280.893,E2 -8280.893} C_VEL
LIN {X 0,Y 452.564,Z 436.244,A -85,B 0,C 180,E1 -8281.783,E2 -8281.783} C_VEL
LIN {X 0,Y 452.629,Z 435.045,A -85,B 0,C 180,E1 -8282.673,E2 -8282.673} C_VEL
LIN {X 0,Y 452.789,Z 432.187,A -85,B 0,C 180,E1 -8284.008,E2 -8284.008} C_VEL
LIN {X 0,Y 452.879,Z 429.538,A -85,B 0,C 180,E1 -8284.899,E2 -8284.899} C_VEL
LIN {X 0,Y 452.913,Z 426.25,A -85,B 0,C 180,E1 -8285.792,E2 -8285.792} C_VEL
LIN {X 0,Y 453.208,Z 421.936,A -85,B 0,C 180,E1 -8286.737,E2 -8286.737} C_VEL
LIN {X 0,Y 453.279,Z 417.369,A -85,B 0,C 180,E1 -8287.576,E2 -8287.576} C_VEL
LIN {X 0,Y 453.576,Z 411.499,A -85,B 0,C 180,E1 -8288.467,E2 -8288.467} C_VEL
LIN {X 0,Y 453.878,Z 404.371,A -85,B 0,C 180,E1 -8289.36,E2 -8289.36} C_VEL
LIN {X 0,Y 454.218,Z 395.605,A -85,B 0,C 180,E1 -8290.252,E2 -8290.252} C_VEL
LIN {X 0,Y 454.589,Z 385.817,A -85,B 0,C 180,E1 -8291.032,E2 -8291.032} C_VEL
LIN {X 0,Y 454.853,Z 375.646,A -85,B 0,C 180,E1 -8291.646,E2 -8291.646} C_VEL
LIN {X 0,Y 455.014,Z 366.49,A -85,B 0,C 180,E1 -8292.066,E2 -8292.066} C_VEL
LIN {X 0,Y 455.235,Z 355.147,A -85,B 0,C 180,E1 -8292.428,E2 -8292.428} C_VEL
LIN {X 0,Y 455.936,Z 290.409,A -85,B 0,C 180,E1 -8293.678,E2 -8293.678} C_VEL
LIN {X 0,Y 453.751,Z 279.308,A -85,B 0,C 180,E1 -8294.008,E2 -8294.008} C_VEL
LIN {X 0,Y 453.889,Z 267.329,A -85,B 0,C 180,E1 -8296.857,E2 -8296.857} C_VEL
LIN {X 0,Y 453.58,Z 263.807,A -85,B 0,C 180,E1 -8297.705,E2 -8297.705} C_VEL
LIN {X 0,Y 453.49,Z 263.809,A -85,B 0,C 180,E1 -8300.884,E2 -8300.884} C_VEL
LIN {X 0,Y 453.498,Z 263.809,A -85,B 0,C 180,E1 -8303.887,E2 -8303.887} C_VEL
LIN {X 0,Y 453.472,Z 263.813,A -85,B 0,C 180,E1 -8306.71,E2 -8306.71} C_VEL
LIN {X 0,Y 453.477,Z 263.81,A -85,B 0,C 180,E1 -8309.785,E2 -8309.785} C_VEL
LIN {X 0,Y 453.492,Z 263.807,A -85,B 0,C 180,E1 -8313.189,E2 -8313.189} C_VEL
LIN {X 0,Y 453.458,Z 263.816,A -85,B 0,C 180,E1 -8316.299,E2 -8316.299} C_VEL
LIN {X 0,Y 453.457,Z 263.81,A -85,B 0,C 180,E1 -8319.455,E2 -8319.455} C_VEL
LIN {X 0,Y 453.465,Z 263.81,A -85,B 0,C 180,E1 -8321.933,E2 -8321.933} C_VEL
LIN {X 0,Y 453.491,Z 263.805,A -85,B 0,C 180,E1 -8325.472,E2 -8325.472} C_VEL
LIN {X 0,Y 453.471,Z 263.81,A -85,B 0,C 180,E1 -8328.208,E2 -8328.208} C_VEL
LIN {X 0,Y 453.458,Z 263.815,A -85,B 0,C 180,E1 -8330.801,E2 -8330.801} C_VEL
LIN {X 0,Y 453.458,Z 263.807,A -85,B 0,C 180,E1 -8333.917,E2 -8333.917} C_VEL
LIN {X 0,Y 453.482,Z 263.81,A -85,B 0,C 180,E1 -8337.151,E2 -8337.151} C_VEL
LIN {X 0,Y 453.481,Z 263.81,A -85,B 0,C 180,E1 -8340.268,E2 -8340.268} C_VEL
LIN {X 0,Y 453.506,Z 263.807,A -85,B 0,C 180,E1 -8343.294,E2 -8343.294} C_VEL
LIN {X 0,Y 453.557,Z 263.903,A -85,B 0,C 180,E1 -8345.468,E2 -8345.468} C_VEL
LIN {X 0,Y 454.912,Z 272.522,A -85,B 0,C 180,E1 -8347.28,E2 -8347.28} C_VEL
LIN {X 0,Y 454.4,Z 286.671,A -85,B 0,C 180,E1 -8350.107,E2 -8350.107} C_VEL
LIN {X 0,Y 453.749,Z 301.939,A -85,B 0,C 180,E1 -8353.117,E2 -8353.117} C_VEL
LIN {X 0,Y 453.338,Z 317.154,A -85,B 0,C 180,E1 -8356.096,E2 -8356.096} C_VEL
LIN {X 0,Y 453.287,Z 318.114,A -85,B 0,C 180,E1 -8356.283,E2 -8356.283} C_VEL
LIN {X 0,Y 455.478,Z 338.712,A -85,B 0,C 180,E1 -8356.671,E2 -8356.671} C_VEL
LIN {X 0,Y 455.083,Z 395.933,A -85,B 0,C 180,E1 -8357.598,E2 -8357.598} C_VEL
LIN {X 0,Y 454.792,Z 406.464,A -85,B 0,C 180,E1 -8357.902,E2 -8357.902} C_VEL
LIN {X 0,Y 454.446,Z 417.746,A -85,B 0,C 180,E1 -8358.402,E2 -8358.402} C_VEL
LIN {X 0,Y 454.141,Z 426.79,A -85,B 0,C 180,E1 -8358.959,E2 -8358.959} C_VEL
LIN {X 0,Y 453.807,Z 435.352,A -85,B 0,C 180,E1 -8359.628,E2 -8359.628} C_VEL
LIN {X 0,Y 453.491,Z 443.42,A -85,B 0,C 180,E1 -8360.41,E2 -8360.41} C_VEL
LIN {X 0,Y 453.258,Z 449.225,A -85,B 0,C 180,E1 -8361.08,E2 -8361.08} C_VEL
LIN {X 0,Y 452.965,Z 455.695,A -85,B 0,C 180,E1 -8361.973,E2 -8361.973} C_VEL
LIN {X 0,Y 452.878,Z 461.08,A -85,B 0,C 180,E1 -8362.868,E2 -8362.868} C_VEL
LIN {X 0,Y 452.657,Z 465.562,A -85,B 0,C 180,E1 -8363.76,E2 -8363.76} C_VEL
LIN {X 0,Y 452.622,Z 469.302,A -85,B 0,C 180,E1 -8364.654,E2 -8364.654} C_VEL
LIN {X 0,Y 452.508,Z 473.544,A -85,B 0,C 180,E1 -8365.992,E2 -8365.992} C_VEL
LIN {X 0,Y 452.535,Z 476.512,A -85,B 0,C 180,E1 -8367.329,E2 -8367.329} C_VEL
LIN {X 0,Y 452.485,Z 477.809,A -85,B 0,C 180,E1 -8368.22,E2 -8368.22} C_VEL
LIN {X 0,Y 452.491,Z 478.63,A -85,B 0,C 180,E1 -8369.11,E2 -8369.11} C_VEL
LIN {X 0,Y 452.471,Z 478.934,A -85,B 0,C 180,E1 -8370,E2 -8370} C_VEL
LIN {X 0,Y 452.475,Z 478.653,A -85,B 0,C 180,E1 -8370.89,E2 -8370.89} C_VEL
LIN {X 0,Y 452.485,Z 477.898,A -85,B 0,C 180,E1 -8371.78,E2 -8371.78} C_VEL
LIN {X 0,Y 452.535,Z 476.67,A -85,B 0,C 180,E1 -8372.67,E2 -8372.67} C_VEL
LIN {X 0,Y 452.546,Z 474.943,A -85,B 0,C 180,E1 -8373.561,E2 -8373.561} C_VEL
LIN {X 0,Y 452.58,Z 471.157,A -85,B 0,C 180,E1 -8374.899,E2 -8374.899} C_VEL
LIN {X 0,Y 452.656,Z 465.992,A -85,B 0,C 180,E1 -8376.239,E2 -8376.239} C_VEL
LIN {X 0,Y 452.888,Z 460.451,A -85,B 0,C 180,E1 -8377.355,E2 -8377.355} C_VEL
LIN {X 0,Y 453.13,Z 453.525,A -85,B 0,C 180,E1 -8378.473,E2 -8378.473} C_VEL
LIN {X 0,Y 453.521,Z 444.57,A -85,B 0,C 180,E1 -8379.589,E2 -8379.589} C_VEL
LIN {X 0,Y 453.882,Z 436.801,A -85,B 0,C 180,E1 -8380.37,E2 -8380.37} C_VEL
LIN {X 0,Y 454.168,Z 430.136,A -85,B 0,C 180,E1 -8380.927,E2 -8380.927} C_VEL
LIN {X 0,Y 454.483,Z 422.02,A -85,B 0,C 180,E1 -8381.484,E2 -8381.484} C_VEL
LIN {X 0,Y 454.78,Z 412.649,A -85,B 0,C 180,E1 -8381.985,E2 -8381.985} C_VEL
LIN {X 0,Y 455.115,Z 403.48,A -85,B 0,C 180,E1 -8382.344,E2 -8382.344} C_VEL
LIN {X 0,Y 455.425,Z 394.014,A -85,B 0,C 180,E1 -8382.59,E2 -8382.59} C_VEL
LIN {X 0,Y 455.678,Z 336.119,A -85,B 0,C 180,E1 -8383.53,E2 -8383.53} C_VEL
LIN {X 0,Y 453.37,Z 317.642,A -85,B 0,C 180,E1 -8383.931,E2 -8383.931} C_VEL
LIN {X 0,Y 453.839,Z 302.737,A -85,B 0,C 180,E1 -8386.856,E2 -8386.856} C_VEL
LIN {X 0,Y 454.505,Z 286.254,A -85,B 0,C 180,E1 -8390.124,E2 -8390.124} C_VEL
LIN {X 0,Y 455.023,Z 273.382,A -85,B 0,C 180,E1 -8392.714,E2 -8392.714} C_VEL
LIN {X 0,Y 454.127,Z 267.043,A -85,B 0,C 180,E1 -8394.064,E2 -8394.064} C_VEL
LIN {X 0,Y 453.526,Z 263.807,A -85,B 0,C 180,E1 -8394.795,E2 -8394.795} C_VEL
LIN {X 0,Y 453.537,Z 263.802,A -85,B 0,C 180,E1 -8397.959,E2 -8397.959} C_VEL
LIN {X 0,Y 453.47,Z 263.81,A -85,B 0,C 180,E1 -8401.524,E2 -8401.524} C_VEL
LIN {X 0,Y 453.488,Z 263.809,A -85,B 0,C 180,E1 -8404.775,E2 -8404.775} C_VEL
LIN {X 0,Y 453.465,Z 263.809,A -85,B 0,C 180,E1 -8408.311,E2 -8408.311} C_VEL
LIN {X 0,Y 453.5,Z 263.804,A -85,B 0,C 180,E1 -8410.608,E2 -8410.608} C_VEL
LIN {X 0,Y 453.467,Z 263.806,A -85,B 0,C 180,E1 -8414.221,E2 -8414.221} C_VEL
LIN {X 0,Y 453.456,Z 263.811,A -85,B 0,C 180,E1 -8417.002,E2 -8417.002} C_VEL
LIN {X 0,Y 453.5,Z 263.81,A -85,B 0,C 180,E1 -8419.408,E2 -8419.408} C_VEL
LIN {X 0,Y 453.458,Z 263.809,A -85,B 0,C 180,E1 -8422.809,E2 -8422.809} C_VEL
LIN {X 0,Y 453.475,Z 263.809,A -85,B 0,C 180,E1 -8426.085,E2 -8426.085} C_VEL
LIN {X 0,Y 453.481,Z 263.805,A -85,B 0,C 180,E1 -8429.239,E2 -8429.239} C_VEL
LIN {X 0,Y 453.514,Z 263.801,A -85,B 0,C 180,E1 -8432.294,E2 -8432.294} C_VEL
LIN {X 0,Y 453.506,Z 263.803,A -85,B 0,C 180,E1 -8435.263,E2 -8435.263} C_VEL
LIN {X 0,Y 453.486,Z 263.801,A -85,B 0,C 180,E1 -8438.413,E2 -8438.413} C_VEL
LIN {X 0,Y 453.528,Z 263.799,A -85,B 0,C 180,E1 -8441.007,E2 -8441.007} C_VEL
LIN {X 0,Y 453.574,Z 263.795,A -85,B 0,C 180,E1 -8443.878,E2 -8443.878} C_VEL
LIN {X 0,Y 453.568,Z 263.796,A -85,B 0,C 180,E1 -8447.469,E2 -8447.469} C_VEL
LIN {X 0,Y 453.594,Z 263.789,A -85,B 0,C 180,E1 -8451.084,E2 -8451.084} C_VEL
LIN {X 0,Y 453.673,Z 263.783,A -85,B 0,C 180,E1 -8453.772,E2 -8453.772} C_VEL
LIN {X 0,Y 453.734,Z 263.772,A -85,B 0,C 180,E1 -8457.334,E2 -8457.334} C_VEL
LIN {X 0,Y 453.82,Z 263.763,A -85,B 0,C 180,E1 -8459.997,E2 -8459.997} C_VEL
LIN {X 0,Y 453.735,Z 263.774,A -85,B 0,C 180,E1 -8462.66,E2 -8462.66} C_VEL
LIN {X 0,Y 453.646,Z 263.787,A -85,B 0,C 180,E1 -8466.223,E2 -8466.223} C_VEL
LIN {X 0,Y 453.582,Z 263.792,A -85,B 0,C 180,E1 -8468.91,E2 -8468.91} C_VEL
LIN {X 0,Y 453.558,Z 263.801,A -85,B 0,C 180,E1 -8472.526,E2 -8472.526} C_VEL
LIN {X 0,Y 453.537,Z 263.8,A -85,B 0,C 180,E1 -8476.193,E2 -8476.193} C_VEL
LIN {X 0,Y 453.508,Z 263.802,A -85,B 0,C 180,E1 -8479.036,E2 -8479.036} C_VEL
LIN {X 0,Y 453.466,Z 263.808,A -85,B 0,C 180,E1 -8481.833,E2 -8481.833} C_VEL
LIN {X 0,Y 453.501,Z 263.806,A -85,B 0,C 180,E1 -8484.731,E2 -8484.731} C_VEL
LIN {X 0,Y 453.518,Z 263.803,A -85,B 0,C 180,E1 -8487.956,E2 -8487.956} C_VEL
LIN {X 0,Y 453.449,Z 263.808,A -85,B 0,C 180,E1 -8491.522,E2 -8491.522} C_VEL
LIN {X 0,Y 453.47,Z 263.806,A -85,B 0,C 180,E1 -8494.774,E2 -8494.774} C_VEL
LIN {X 0,Y 453.444,Z 263.815,A -85,B 0,C 180,E1 -8498.308,E2 -8498.308} C_VEL
LIN {X 0,Y 453.471,Z 263.808,A -85,B 0,C 180,E1 -8501.786,E2 -8501.786} C_VEL
LIN {X 0,Y 453.469,Z 263.81,A -85,B 0,C 180,E1 -8504.527,E2 -8504.527} C_VEL
LIN {X 0,Y 453.471,Z 263.809,A -85,B 0,C 180,E1 -8508.059,E2 -8508.059} C_VEL
LIN {X 0,Y 453.505,Z 263.81,A -85,B 0,C 180,E1 -8510.785,E2 -8510.785} C_VEL
LIN {X 0,Y 453.429,Z 263.816,A -85,B 0,C 180,E1 -8513.915,E2 -8513.915} C_VEL
LIN {X 0,Y 453.519,Z 263.882,A -85,B 0,C 180,E1 -8515.722,E2 -8515.722} C_VEL
LIN {X 0,Y 453.766,Z 270.011,A -85,B 0,C 180,E1 -8517.174,E2 -8517.174} C_VEL
LIN {X 0,Y 453.601,Z 278.487,A -85,B 0,C 180,E1 -8519.152,E2 -8519.152} C_VEL
LIN {X 0,Y 456.037,Z 291.329,A -85,B 0,C 180,E1 -8519.447,E2 -8519.447} C_VEL
LIN {X 0,Y 455.504,Z 354.693,A -85,B 0,C 180,E1 -8520.478,E2 -8520.478} C_VEL
LIN {X 0,Y 455.351,Z 364.309,A -85,B 0,C 180,E1 -8520.752,E2 -8520.752} C_VEL
LIN {X 0,Y 455.126,Z 375.058,A -85,B 0,C 180,E1 -8521.211,E2 -8521.211} C_VEL
LIN {X 0,Y 454.783,Z 386.364,A -85,B 0,C 180,E1 -8521.906,E2 -8521.906} C_VEL
LIN {X 0,Y 454.452,Z 395.07,A -85,B 0,C 180,E1 -8522.608,E2 -8522.608} C_VEL
LIN {X 0,Y 454.077,Z 402.381,A -85,B 0,C 180,E1 -8523.33,E2 -8523.33} C_VEL
LIN {X 0,Y 453.759,Z 409.229,A -85,B 0,C 180,E1 -8524.151,E2 -8524.151} C_VEL
LIN {X 0,Y 453.469,Z 415.232,A -85,B 0,C 180,E1 -8525.018,E2 -8525.018} C_VEL
LIN {X 0,Y 453.246,Z 420.865,A -85,B 0,C 180,E1 -8526.006,E2 -8526.006} C_VEL
LIN {X 0,Y 452.994,Z 425.232,A -85,B 0,C 180,E1 -8526.937,E2 -8526.937} C_VEL
LIN {X 0,Y 452.812,Z 429.315,A -85,B 0,C 180,E1 -8528.019,E2 -8528.019} C_VEL
LIN {X 0,Y 452.068,Z 431.546,A -85,B 0,C 180,E1 -8528.707,E2 -8528.707} C_VEL
LIN {X 0,Y 449.08,Z 434.517,A -85,B 0,C 180,E1 -8529.849,E2 -8529.849} C_VEL
LIN {X 0,Y 446.092,Z 436.506,A -85,B 0,C 180,E1 -8531.037,E2 -8531.037} C_VEL
LIN {X 0,Y 445.362,Z 437.127,A -85,B 0,C 180,E1 -8531.788,E2 -8531.788} C_VEL
LIN {X 0,Y 445.338,Z 437.497,A -85,B 0,C 180,E1 -8532.552,E2 -8532.552} C_VEL
LIN {X 0,Y 445.41,Z 437.081,A -85,B 0,C 180,E1 -8534.242,E2 -8534.242} C_VEL
LIN {X 0,Y 445.431,Z 435.792,A -85,B 0,C 180,E1 -8535.378,E2 -8535.378} C_VEL
LIN {X 0,Y 445.534,Z 433.009,A -85,B 0,C 180,E1 -8536.778,E2 -8536.778} C_VEL
LIN {X 0,Y 445.73,Z 428.932,A -85,B 0,C 180,E1 -8538.172,E2 -8538.172} C_VEL
LIN {X 0,Y 445.848,Z 425.393,A -85,B 0,C 180,E1 -8539.096,E2 -8539.096} C_VEL
LIN {X 0,Y 446.055,Z 421.103,A -85,B 0,C 180,E1 -8540.02,E2 -8540.02} C_VEL
LIN {X 0,Y 446.3,Z 415.941,A -85,B 0,C 180,E1 -8540.94,E2 -8540.94} C_VEL
LIN {X 0,Y 446.572,Z 409.72,A -85,B 0,C 180,E1 -8541.857,E2 -8541.857} C_VEL
LIN {X 0,Y 446.838,Z 403.271,A -85,B 0,C 180,E1 -8542.648,E2 -8542.648} C_VEL
LIN {X 0,Y 447.131,Z 396.495,A -85,B 0,C 180,E1 -8543.343,E2 -8543.343} C_VEL
LIN {X 0,Y 447.446,Z 388.387,A -85,B 0,C 180,E1 -8544.027,E2 -8544.027} C_VEL
LIN {X 0,Y 447.76,Z 379.953,A -85,B 0,C 180,E1 -8544.596,E2 -8544.596} C_VEL
LIN {X 0,Y 447.93,Z 371.393,A -85,B 0,C 180,E1 -8545.05,E2 -8545.05} C_VEL
LIN {X 0,Y 448.139,Z 361.126,A -85,B 0,C 180,E1 -8545.446,E2 -8545.446} C_VEL
LIN {X 0,Y 448.337,Z 347.11,A -85,B 0,C 180,E1 -8545.758,E2 -8545.758} C_VEL
LIN {X 0,Y 448.621,Z 290.947,A -85,B 0,C 180,E1 -8546.66,E2 -8546.66} C_VEL
LIN {X 0,Y 446.39,Z 278.744,A -85,B 0,C 180,E1 -8546.926,E2 -8546.926} C_VEL
LIN {X 0,Y 446.701,Z 266.141,A -85,B 0,C 180,E1 -8550,E2 -8550} C_VEL
LIN {X 0,Y 446.608,Z 264.667,A -85,B 0,C 180,E1 -8550.395,E2 -8550.395} C_VEL
LIN {X 0,Y 446.672,Z 264.656,A -85,B 0,C 180,E1 -8552.706,E2 -8552.706} C_VEL
LIN {X 0,Y 446.603,Z 264.663,A -85,B 0,C 180,E1 -8556.324,E2 -8556.324} C_VEL
LIN {X 0,Y 446.501,Z 264.68,A -85,B 0,C 180,E1 -8559.056,E2 -8559.056} C_VEL
LIN {X 0,Y 446.485,Z 264.678,A -85,B 0,C 180,E1 -8562.731,E2 -8562.731} C_VEL
LIN {X 0,Y 446.454,Z 264.681,A -85,B 0,C 180,E1 -8566.461,E2 -8566.461} C_VEL
LIN {X 0,Y 446.434,Z 264.69,A -85,B 0,C 180,E1 -8569.305,E2 -8569.305} C_VEL
LIN {X 0,Y 446.382,Z 264.69,A -85,B 0,C 180,E1 -8572.202,E2 -8572.202} C_VEL
LIN {X 0,Y 446.404,Z 264.691,A -85,B 0,C 180,E1 -8575.156,E2 -8575.156} C_VEL
LIN {X 0,Y 446.408,Z 264.687,A -85,B 0,C 180,E1 -8578.184,E2 -8578.184} C_VEL
LIN {X 0,Y 446.384,Z 264.694,A -85,B 0,C 180,E1 -8581.303,E2 -8581.303} C_VEL
LIN {X 0,Y 446.398,Z 264.688,A -85,B 0,C 180,E1 -8584.526,E2 -8584.526} C_VEL
LIN {X 0,Y 446.382,Z 264.692,A -85,B 0,C 180,E1 -8588.081,E2 -8588.081} C_VEL
LIN {X 0,Y 446.385,Z 264.694,A -85,B 0,C 180,E1 -8591.396,E2 -8591.396} C_VEL
LIN {X 0,Y 446.427,Z 264.686,A -85,B 0,C 180,E1 -8595.107,E2 -8595.107} C_VEL
LIN {X 0,Y 446.407,Z 264.687,A -85,B 0,C 180,E1 -8598.612,E2 -8598.612} C_VEL
LIN {X 0,Y 446.394,Z 264.694,A -85,B 0,C 180,E1 -8601.925,E2 -8601.925} C_VEL
LIN {X 0,Y 446.406,Z 264.691,A -85,B 0,C 180,E1 -8605.48,E2 -8605.48} C_VEL
LIN {X 0,Y 446.401,Z 264.688,A -85,B 0,C 180,E1 -8608.703,E2 -8608.703} C_VEL
LIN {X 0,Y 446.437,Z 264.691,A -85,B 0,C 180,E1 -8611.833,E2 -8611.833} C_VEL
LIN {X 0,Y 446.428,Z 264.685,A -85,B 0,C 180,E1 -8614.85,E2 -8614.85} C_VEL
LIN {X 0,Y 446.44,Z 264.686,A -85,B 0,C 180,E1 -8618.249,E2 -8618.249} C_VEL
LIN {X 0,Y 446.443,Z 264.687,A -85,B 0,C 180,E1 -8621.652,E2 -8621.652} C_VEL
LIN {X 0,Y 446.517,Z 264.835,A -85,B 0,C 180,E1 -8622.957,E2 -8622.957} C_VEL
LIN {X 0,Y 446.432,Z 274.853,A -85,B 0,C 180,E1 -8625.415,E2 -8625.415} C_VEL
LIN {X 0,Y 446.402,Z 278.335,A -85,B 0,C 180,E1 -8626.264,E2 -8626.264} C_VEL
LIN {X 0,Y 448.472,Z 292.248,A -85,B 0,C 180,E1 -8626.584,E2 -8626.584} C_VEL
LIN {X 0,Y 447.841,Z 355.422,A -85,B 0,C 180,E1 -8627.772,E2 -8627.772} C_VEL
LIN {X 0,Y 447.65,Z 365.9,A -85,B 0,C 180,E1 -8628.112,E2 -8628.112} C_VEL
LIN {X 0,Y 447.392,Z 375.679,A -85,B 0,C 180,E1 -8628.564,E2 -8628.564} C_VEL
LIN {X 0,Y 447.204,Z 386.631,A -85,B 0,C 180,E1 -8629.248,E2 -8629.248} C_VEL
LIN {X 0,Y 446.864,Z 396.151,A -85,B 0,C 180,E1 -8630.041,E2 -8630.041} C_VEL
LIN {X 0,Y 446.62,Z 402.866,A -85,B 0,C 180,E1 -8630.721,E2 -8630.721} C_VEL
LIN {X 0,Y 446.307,Z 410.271,A -85,B 0,C 180,E1 -8631.628,E2 -8631.628} C_VEL
LIN {X 0,Y 446.106,Z 416.385,A -85,B 0,C 180,E1 -8632.535,E2 -8632.535} C_VEL
LIN {X 0,Y 446.029,Z 420.836,A -85,B 0,C 180,E1 -8633.323,E2 -8633.323} C_VEL
LIN {X 0,Y 445.833,Z 424.708,A -85,B 0,C 180,E1 -8634.122,E2 -8634.122} C_VEL
LIN {X 0,Y 445.663,Z 429.899,A -85,B 0,C 180,E1 -8635.481,E2 -8635.481} C_VEL
LIN {X 0,Y 445.574,Z 433.691,A -85,B 0,C 180,E1 -8636.838,E2 -8636.838} C_VEL
LIN {X 0,Y 445.434,Z 436.082,A -85,B 0,C 180,E1 -8638.195,E2 -8638.195} C_VEL
LIN {X 0,Y 445.403,Z 437.056,A -85,B 0,C 180,E1 -8639.099,E2 -8639.099} C_VEL
LIN {X 0,Y 445.41,Z 437.439,A -85,B 0,C 180,E1 -8640.003,E2 -8640.003} C_VEL
LIN {X 0,Y 445.434,Z 437.279,A -85,B 0,C 180,E1 -8640.907,E2 -8640.907} C_VEL
LIN {X 0,Y 445.477,Z 436.615,A -85,B 0,C 180,E1 -8641.811,E2 -8641.811} C_VEL
LIN {X 0,Y 445.555,Z 435.442,A -85,B 0,C 180,E1 -8642.715,E2 -8642.715} C_VEL
